gfCNCPoint6[12068] = {X 364.4434, Y 8.9212, Z -8.0000, A 0.000, B 0.000, C 0.000 }
gfCNCPoint6[12069] = {X 365.7826, Y 10.9065, Z -8.0000, A 0.000, B 0.000, C 0.000 }
gfCNCPoint6[12070] = {X 366.9214, Y 13.0132, Z -8.0000, A 0.000, B 0.000, C 0.000 }
gfCNCPoint6[12071] = {X 367.8488, Y 15.2212, Z -8.0000, A 0.000, B 0.000, C 0.000 }
gfCNCPoint6[12072] = {X 368.5559, Y 17.5092, Z -8.0000, A 0.000, B 0.000, C 0.000 }
gfCNCPoint6[12073] = {X 369.0331, Y 19.7784, Z -8.0000, A 0.000, B 0.000, C 0.000 }
gfCNCPoint6[12074] = {X 369.3408, Y 22.0767, Z -8.0000, A 0.000, B 0.000, C 0.000 }
gfCNCPoint6[12075] = {X 369.4773, Y 24.3915, Z -8.0000, A 0.000, B 0.000, C 0.000 }
gfCNCPoint6[12076] = {X 369.4418, Y 26.7100, Z -8.0000, A 0.000, B 0.000, C 0.000 }
gfCNCPoint6[12077] = {X 369.2346, Y 29.0196, Z -8.0000, A 0.000, B 0.000, C 0.000 }
gfCNCPoint6[12078] = {X 368.8568, Y 31.3074, Z -8.0000, A 0.000, B 0.000, C 0.000 }
gfCNCPoint6[12079] = {X 368.3394, Y 33.3846, Z -8.0000, A 0.000, B 0.000, C 0.000 }
gfCNCPoint6[12080] = {X 367.6406, Y 35.4079, Z -8.0000, A 0.000, B 0.000, C 0.000 }
gfCNCPoint6[12081] = {X 366.7658, Y 37.3616, Z -8.0000, A 0.000, B 0.000, C 0.000 }
gfCNCPoint6[12082] = {X 365.7220, Y 39.2305, Z -8.0000, A 0.000, B 0.000, C 0.000 }
gfCNCPoint6[12083] = {X 364.5172, Y 40.9999, Z -8.0000, A 0.000, B 0.000, C 0.000 }
gfCNCPoint6[12084] = {X 364.4579, Y 41.0809, Z -8.0000, A 0.000, B 0.000, C 0.000 }
gfCNCPoint6[12085] = {X 367.7503, Y 43.4906, Z -8.0000, A 0.000, B 0.000, C 0.000 }
gfCNCPoint6[12086] = {X 367.7503, Y 43.4906, Z -5.0000, A 0.000, B 0.000, C 0.000 }
gfCNCPoint6[12087] = {X 367.7503, Y 43.4906, Z 11.0000, A 0.000, B 0.000, C 0.000 }
gfCNCPoint6[12088] = {X 606.0426, Y 42.9003, Z 11.0000, A 0.000, B 0.000, C 0.000 }
gfCNCPoint6[12089] = {X 606.0426, Y 42.9003, Z -5.0000, A 0.000, B 0.000, C 0.000 }
gfCNCPoint6[12090] = {X 606.0426, Y 42.9003, Z -8.0000, A 0.000, B 0.000, C 0.000 }
gfCNCPoint6[12091] = {X 603.6967, Y 47.0765, Z -8.0000, A 0.000, B 0.000, C 0.000 }
gfCNCPoint6[12092] = {X 603.6312, Y 47.1891, Z -8.0000, A 0.000, B 0.000, C 0.000 }
gfCNCPoint6[12093] = {X 603.5623, Y 47.2995, Z -8.0000, A 0.000, B 0.000, C 0.000 }
gfCNCPoint6[12094] = {X 603.0359, Y 47.9599, Z -8.0000, A 0.000, B 0.000, C 0.000 }
gfCNCPoint6[12095] = {X 602.3890, Y 48.5029, Z -8.0000, A 0.000, B 0.000, C 0.000 }
gfCNCPoint6[12096] = {X 601.6473, Y 48.9069, Z -8.0000, A 0.000, B 0.000, C 0.000 }
gfCNCPoint6[12097] = {X 600.8403, Y 49.1559, Z -8.0000, A 0.000, B 0.000, C 0.000 }
gfCNCPoint6[12098] = {X 600.0000, Y 49.2400, Z -8.0000, A 0.000, B 0.000, C 0.000 }
gfCNCPoint6[12099] = {X 593.5565, Y 49.2400, Z -8.0000, A 0.000, B 0.000, C 0.000 }
gfCNCPoint6[12100] = {X 592.6130, Y 49.1337, Z -8.0000, A 0.000, B 0.000, C 0.000 }
gfCNCPoint6[12101] = {X 591.7169, Y 48.8201, Z -8.0000, A 0.000, B 0.000, C 0.000 }
gfCNCPoint6[12102] = {X 590.9129, Y 48.3150, Z -8.0000, A 0.000, B 0.000, C 0.000 }
gfCNCPoint6[12103] = {X 590.2416, Y 47.6436, Z -8.0000, A 0.000, B 0.000, C 0.000 }
gfCNCPoint6[12104] = {X 589.7364, Y 46.8397, Z -8.0000, A 0.000, B 0.000, C 0.000 }
gfCNCPoint6[12105] = {X 589.4228, Y 45.9435, Z -8.0000, A 0.000, B 0.000, C 0.000 }
gfCNCPoint6[12106] = {X 589.3165, Y 45.0000, Z -8.0000, A 0.000, B 0.000, C 0.000 }
gfCNCPoint6[12107] = {X 589.3165, Y 44.0651, Z -8.0000, A 0.000, B 0.000, C 0.000 }
gfCNCPoint6[12108] = {X 589.4202, Y 43.1448, Z -8.0000, A 0.000, B 0.000, C 0.000 }
gfCNCPoint6[12109] = {X 589.7196, Y 42.2684, Z -8.0000, A 0.000, B 0.000, C 0.000 }
gfCNCPoint6[12110] = {X 590.2007, Y 41.4770, Z -8.0000, A 0.000, B 0.000, C 0.000 }
gfCNCPoint6[12111] = {X 590.8409, Y 40.8078, Z -8.0000, A 0.000, B 0.000, C 0.000 }
gfCNCPoint6[12112] = {X 590.8418, Y 33.1230, Z -8.0000, A 0.000, B 0.000, C 0.000 }
gfCNCPoint6[12113] = {X 585.3714, Y 46.6218, Z -8.0000, A 0.000, B 0.000, C 0.000 }
gfCNCPoint6[12114] = {X 585.0085, Y 47.3114, Z -8.0000, A 0.000, B 0.000, C 0.000 }
gfCNCPoint6[12115] = {X 584.5255, Y 47.9228, Z -8.0000, A 0.000, B 0.000, C 0.000 }
gfCNCPoint6[12116] = {X 583.9387, Y 48.4356, Z -8.0000, A 0.000, B 0.000, C 0.000 }
gfCNCPoint6[12117] = {X 583.2680, Y 48.8323, Z -8.0000, A 0.000, B 0.000, C 0.000 }
gfCNCPoint6[12118] = {X 582.3418, Y 49.1460, Z -8.0000, A 0.000, B 0.000, C 0.000 }
gfCNCPoint6[12119] = {X 581.3682, Y 49.2391, Z -8.0000, A 0.000, B 0.000, C 0.000 }
gfCNCPoint6[12120] = {X 580.3993, Y 49.1068, Z -8.0000, A 0.000, B 0.000, C 0.000 }
gfCNCPoint6[12121] = {X 579.4864, Y 48.7559, Z -8.0000, A 0.000, B 0.000, C 0.000 }
gfCNCPoint6[12122] = {X 578.6782, Y 48.2052, Z -8.0000, A 0.000, B 0.000, C 0.000 }
gfCNCPoint6[12123] = {X 578.0177, Y 47.4840, Z -8.0000, A 0.000, B 0.000, C 0.000 }
gfCNCPoint6[12124] = {X 577.5400, Y 46.6307, Z -8.0000, A 0.000, B 0.000, C 0.000 }
gfCNCPoint6[12125] = {X 571.9402, Y 32.9378, Z -8.0000, A 0.000, B 0.000, C 0.000 }
gfCNCPoint6[12126] = {X 571.9404, Y 40.8087, Z -8.0000, A 0.000, B 0.000, C 0.000 }
gfCNCPoint6[12127] = {X 571.9716, Y 40.8346, Z -8.0000, A 0.000, B 0.000, C 0.000 }
gfCNCPoint6[12128] = {X 572.5965, Y 41.4929, Z -8.0000, A 0.000, B 0.000, C 0.000 }
gfCNCPoint6[12129] = {X 573.0669, Y 42.2692, Z -8.0000, A 0.000, B 0.000, C 0.000 }
gfCNCPoint6[12130] = {X 573.3613, Y 43.1278, Z -8.0000, A 0.000, B 0.000, C 0.000 }
gfCNCPoint6[12131] = {X 573.4663, Y 44.0294, Z -8.0000, A 0.000, B 0.000, C 0.000 }
gfCNCPoint6[12132] = {X 573.4664, Y 45.0000, Z -8.0000, A 0.000, B 0.000, C 0.000 }
gfCNCPoint6[12133] = {X 573.3601, Y 45.9435, Z -8.0000, A 0.000, B 0.000, C 0.000 }
gfCNCPoint6[12134] = {X 573.0465, Y 46.8397, Z -8.0000, A 0.000, B 0.000, C 0.000 }
gfCNCPoint6[12135] = {X 572.5414, Y 47.6436, Z -8.0000, A 0.000, B 0.000, C 0.000 }
gfCNCPoint6[12136] = {X 571.8700, Y 48.3150, Z -8.0000, A 0.000, B 0.000, C 0.000 }
gfCNCPoint6[12137] = {X 571.0661, Y 48.8201, Z -8.0000, A 0.000, B 0.000, C 0.000 }
gfCNCPoint6[12138] = {X 570.1699, Y 49.1337, Z -8.0000, A 0.000, B 0.000, C 0.000 }
gfCNCPoint6[12139] = {X 569.2264, Y 49.2400, Z -8.0000, A 0.000, B 0.000, C 0.000 }
gfCNCPoint6[12140] = {X 562.4443, Y 49.2400, Z -8.0000, A 0.000, B 0.000, C 0.000 }
gfCNCPoint6[12141] = {X 561.5008, Y 49.1337, Z -8.0000, A 0.000, B 0.000, C 0.000 }
gfCNCPoint6[12142] = {X 560.6046, Y 48.8201, Z -8.0000, A 0.000, B 0.000, C 0.000 }
gfCNCPoint6[12143] = {X 559.8007, Y 48.3150, Z -8.0000, A 0.000, B 0.000, C 0.000 }
gfCNCPoint6[12144] = {X 559.1293, Y 47.6436, Z -8.0000, A 0.000, B 0.000, C 0.000 }
gfCNCPoint6[12145] = {X 558.6242, Y 46.8397, Z -8.0000, A 0.000, B 0.000, C 0.000 }
gfCNCPoint6[12146] = {X 558.3106, Y 45.9435, Z -8.0000, A 0.000, B 0.000, C 0.000 }
gfCNCPoint6[12147] = {X 558.2043, Y 45.0000, Z -8.0000, A 0.000, B 0.000, C 0.000 }
gfCNCPoint6[12148] = {X 558.2043, Y 44.0652, Z -8.0000, A 0.000, B 0.000, C 0.000 }
gfCNCPoint6[12149] = {X 558.3078, Y 43.1444, Z -8.0000, A 0.000, B 0.000, C 0.000 }
gfCNCPoint6[12150] = {X 558.6075, Y 42.2677, Z -8.0000, A 0.000, B 0.000, C 0.000 }
gfCNCPoint6[12151] = {X 559.0893, Y 41.4762, Z -8.0000, A 0.000, B 0.000, C 0.000 }
gfCNCPoint6[12152] = {X 559.7306, Y 40.8074, Z -8.0000, A 0.000, B 0.000, C 0.000 }
gfCNCPoint6[12153] = {X 559.7310, Y 9.1922, Z -8.0000, A 0.000, B 0.000, C 0.000 }
gfCNCPoint6[12154] = {X 559.0934, Y 8.5319, Z -8.0000, A 0.000, B 0.000, C 0.000 }
gfCNCPoint6[12155] = {X 558.6128, Y 7.7499, Z -8.0000, A 0.000, B 0.000, C 0.000 }
gfCNCPoint6[12156] = {X 558.3118, Y 6.8827, Z -8.0000, A 0.000, B 0.000, C 0.000 }
gfCNCPoint6[12157] = {X 558.2045, Y 5.9711, Z -8.0000, A 0.000, B 0.000, C 0.000 }
gfCNCPoint6[12158] = {X 558.2043, Y 5.0000, Z -8.0000, A 0.000, B 0.000, C 0.000 }
gfCNCPoint6[12159] = {X 558.3106, Y 4.0565, Z -8.0000, A 0.000, B 0.000, C 0.000 }
gfCNCPoint6[12160] = {X 558.6242, Y 3.1603, Z -8.0000, A 0.000, B 0.000, C 0.000 }
gfCNCPoint6[12161] = {X 559.1293, Y 2.3564, Z -8.0000, A 0.000, B 0.000, C 0.000 }
gfCNCPoint6[12162] = {X 559.8007, Y 1.6850, Z -8.0000, A 0.000, B 0.000, C 0.000 }
gfCNCPoint6[12163] = {X 560.6046, Y 1.1799, Z -8.0000, A 0.000, B 0.000, C 0.000 }
gfCNCPoint6[12164] = {X 561.5008, Y 0.8663, Z -8.0000, A 0.000, B 0.000, C 0.000 }
gfCNCPoint6[12165] = {X 562.4443, Y 0.7600, Z -8.0000, A 0.000, B 0.000, C 0.000 }
gfCNCPoint6[12166] = {X 570.9376, Y 0.7600, Z -8.0000, A 0.000, B 0.000, C 0.000 }
gfCNCPoint6[12167] = {X 571.8810, Y 0.8663, Z -8.0000, A 0.000, B 0.000, C 0.000 }
gfCNCPoint6[12168] = {X 572.7772, Y 1.1799, Z -8.0000, A 0.000, B 0.000, C 0.000 }
gfCNCPoint6[12169] = {X 573.5812, Y 1.6850, Z -8.0000, A 0.000, B 0.000, C 0.000 }
gfCNCPoint6[12170] = {X 574.2525, Y 2.3564, Z -8.0000, A 0.000, B 0.000, C 0.000 }
gfCNCPoint6[12171] = {X 574.7577, Y 3.1603, Z -8.0000, A 0.000, B 0.000, C 0.000 }
gfCNCPoint6[12172] = {X 575.0712, Y 4.0565, Z -8.0000, A 0.000, B 0.000, C 0.000 }
gfCNCPoint6[12173] = {X 575.1776, Y 5.0000, Z -8.0000, A 0.000, B 0.000, C 0.000 }
gfCNCPoint6[12174] = {X 575.1776, Y 5.9343, Z -8.0000, A 0.000, B 0.000, C 0.000 }
gfCNCPoint6[12175] = {X 575.1024, Y 6.7286, Z -8.0000, A 0.000, B 0.000, C 0.000 }
gfCNCPoint6[12176] = {X 574.8798, Y 7.4948, Z -8.0000, A 0.000, B 0.000, C 0.000 }
gfCNCPoint6[12177] = {X 574.5176, Y 8.2058, Z -8.0000, A 0.000, B 0.000, C 0.000 }
gfCNCPoint6[12178] = {X 581.1908, Y 24.5801, Z -8.0000, A 0.000, B 0.000, C 0.000 }
gfCNCPoint6[12179] = {X 587.9344, Y 8.0873, Z -8.0000, A 0.000, B 0.000, C 0.000 }
gfCNCPoint6[12180] = {X 587.6157, Y 7.4195, Z -8.0000, A 0.000, B 0.000, C 0.000 }
gfCNCPoint6[12181] = {X 587.4179, Y 6.7064, Z -8.0000, A 0.000, B 0.000, C 0.000 }
gfCNCPoint6[12182] = {X 587.3471, Y 5.9698, Z -8.0000, A 0.000, B 0.000, C 0.000 }
gfCNCPoint6[12183] = {X 587.3470, Y 5.0000, Z -8.0000, A 0.000, B 0.000, C 0.000 }
gfCNCPoint6[12184] = {X 587.4533, Y 4.0565, Z -8.0000, A 0.000, B 0.000, C 0.000 }
gfCNCPoint6[12185] = {X 587.7668, Y 3.1603, Z -8.0000, A 0.000, B 0.000, C 0.000 }
gfCNCPoint6[12186] = {X 588.2720, Y 2.3564, Z -8.0000, A 0.000, B 0.000, C 0.000 }
gfCNCPoint6[12187] = {X 588.9434, Y 1.6850, Z -8.0000, A 0.000, B 0.000, C 0.000 }
gfCNCPoint6[12188] = {X 589.7473, Y 1.1799, Z -8.0000, A 0.000, B 0.000, C 0.000 }
gfCNCPoint6[12189] = {X 590.6435, Y 0.8663, Z -8.0000, A 0.000, B 0.000, C 0.000 }
gfCNCPoint6[12190] = {X 591.5870, Y 0.7600, Z -8.0000, A 0.000, B 0.000, C 0.000 }
gfCNCPoint6[12191] = {X 600.0000, Y 0.7600, Z -8.0000, A 0.000, B 0.000, C 0.000 }
gfCNCPoint6[12192] = {X 600.8403, Y 0.8441, Z -8.0000, A 0.000, B 0.000, C 0.000 }
gfCNCPoint6[12193] = {X 601.6473, Y 1.0931, Z -8.0000, A 0.000, B 0.000, C 0.000 }
gfCNCPoint6[12194] = {X 602.3890, Y 1.4971, Z -8.0000, A 0.000, B 0.000, C 0.000 }
gfCNCPoint6[12195] = {X 603.0359, Y 2.0401, Z -8.0000, A 0.000, B 0.000, C 0.000 }
gfCNCPoint6[12196] = {X 603.5623, Y 2.7005, Z -8.0000, A 0.000, B 0.000, C 0.000 }
gfCNCPoint6[12197] = {X 603.6312, Y 2.8109, Z -8.0000, A 0.000, B 0.000, C 0.000 }
gfCNCPoint6[12198] = {X 603.6967, Y 2.9235, Z -8.0000, A 0.000, B 0.000, C 0.000 }
gfCNCPoint6[12199] = {X 607.8224, Y 10.2681, Z -8.0000, A 0.000, B 0.000, C 0.000 }
gfCNCPoint6[12200] = {X 607.8224, Y 10.2681, Z -5.0000, A 0.000, B 0.000, C 0.000 }
gfCNCPoint6[12201] = {X 607.8224, Y 10.2681, Z 11.0000, A 0.000, B 0.000, C 0.000 }
gfCNCPoint6[12202] = {X 607.6967, Y 39.1575, Z 11.0000, A 0.000, B 0.000, C 0.000 }
gfCNCPoint6[12203] = {X 607.6967, Y 39.1575, Z -5.0000, A 0.000, B 0.000, C 0.000 }
gfCNCPoint6[12204] = {X 607.6967, Y 39.1575, Z -8.0000, A 0.000, B 0.000, C 0.000 }
gfCNCPoint6[12205] = {X 603.6967, Y 46.9079, Z -8.0000, A 0.000, B 0.000, C 0.000 }
gfCNCPoint6[12206] = {X 603.6001, Y 47.0845, Z -8.0000, A 0.000, B 0.000, C 0.000 }
gfCNCPoint6[12207] = {X 603.4951, Y 47.2561, Z -8.0000, A 0.000, B 0.000, C 0.000 }
gfCNCPoint6[12208] = {X 602.9786, Y 47.9041, Z -8.0000, A 0.000, B 0.000, C 0.000 }
gfCNCPoint6[12209] = {X 602.3439, Y 48.4368, Z -8.0000, A 0.000, B 0.000, C 0.000 }
gfCNCPoint6[12210] = {X 601.6163, Y 48.8332, Z -8.0000, A 0.000, B 0.000, C 0.000 }
gfCNCPoint6[12211] = {X 600.8245, Y 49.0775, Z -8.0000, A 0.000, B 0.000, C 0.000 }
gfCNCPoint6[12212] = {X 600.0000, Y 49.1600, Z -8.0000, A 0.000, B 0.000, C 0.000 }
gfCNCPoint6[12213] = {X 593.5565, Y 49.1600, Z -8.0000, A 0.000, B 0.000, C 0.000 }
gfCNCPoint6[12214] = {X 592.6308, Y 49.0557, Z -8.0000, A 0.000, B 0.000, C 0.000 }
gfCNCPoint6[12215] = {X 591.7516, Y 48.7480, Z -8.0000, A 0.000, B 0.000, C 0.000 }
gfCNCPoint6[12216] = {X 590.9628, Y 48.2524, Z -8.0000, A 0.000, B 0.000, C 0.000 }
gfCNCPoint6[12217] = {X 590.3041, Y 47.5937, Z -8.0000, A 0.000, B 0.000, C 0.000 }
gfCNCPoint6[12218] = {X 589.8085, Y 46.8050, Z -8.0000, A 0.000, B 0.000, C 0.000 }
gfCNCPoint6[12219] = {X 589.5008, Y 45.9257, Z -8.0000, A 0.000, B 0.000, C 0.000 }
gfCNCPoint6[12220] = {X 589.3965, Y 45.0000, Z -8.0000, A 0.000, B 0.000, C 0.000 }
gfCNCPoint6[12221] = {X 589.3965, Y 44.0654, Z -8.0000, A 0.000, B 0.000, C 0.000 }
gfCNCPoint6[12222] = {X 589.5003, Y 43.1532, Z -8.0000, A 0.000, B 0.000, C 0.000 }
gfCNCPoint6[12223] = {X 589.8000, Y 42.2855, Z -8.0000, A 0.000, B 0.000, C 0.000 }
gfCNCPoint6[12224] = {X 590.2812, Y 41.5037, Z -8.0000, A 0.000, B 0.000, C 0.000 }
gfCNCPoint6[12225] = {X 590.9209, Y 40.8452, Z -8.0000, A 0.000, B 0.000, C 0.000 }
gfCNCPoint6[12226] = {X 590.9218, Y 32.7125, Z -8.0000, A 0.000, B 0.000, C 0.000 }
gfCNCPoint6[12227] = {X 585.2975, Y 46.5912, Z -8.0000, A 0.000, B 0.000, C 0.000 }
gfCNCPoint6[12228] = {X 584.9414, Y 47.2678, Z -8.0000, A 0.000, B 0.000, C 0.000 }
gfCNCPoint6[12229] = {X 584.4675, Y 47.8677, Z -8.0000, A 0.000, B 0.000, C 0.000 }
gfCNCPoint6[12230] = {X 583.8918, Y 48.3708, Z -8.0000, A 0.000, B 0.000, C 0.000 }
gfCNCPoint6[12231] = {X 583.2338, Y 48.7600, Z -8.0000, A 0.000, B 0.000, C 0.000 }
gfCNCPoint6[12232] = {X 582.3250, Y 49.0678, Z -8.0000, A 0.000, B 0.000, C 0.000 }
gfCNCPoint6[12233] = {X 581.3699, Y 49.1592, Z -8.0000, A 0.000, B 0.000, C 0.000 }
gfCNCPoint6[12234] = {X 580.4192, Y 49.0293, Z -8.0000, A 0.000, B 0.000, C 0.000 }
gfCNCPoint6[12235] = {X 579.5236, Y 48.6850, Z -8.0000, A 0.000, B 0.000, C 0.000 }
gfCNCPoint6[12236] = {X 578.7306, Y 48.1448, Z -8.0000, A 0.000, B 0.000, C 0.000 }
gfCNCPoint6[12237] = {X 578.0826, Y 47.4372, Z -8.0000, A 0.000, B 0.000, C 0.000 }
gfCNCPoint6[12238] = {X 577.6138, Y 46.5999, Z -8.0000, A 0.000, B 0.000, C 0.000 }
gfCNCPoint6[12239] = {X 571.8602, Y 32.5308, Z -8.0000, A 0.000, B 0.000, C 0.000 }
gfCNCPoint6[12240] = {X 571.8604, Y 40.8463, Z -8.0000, A 0.000, B 0.000, C 0.000 }
gfCNCPoint6[12241] = {X 571.9201, Y 40.8958, Z -8.0000, A 0.000, B 0.000, C 0.000 }
gfCNCPoint6[12242] = {X 572.5331, Y 41.5417, Z -8.0000, A 0.000, B 0.000, C 0.000 }
gfCNCPoint6[12243] = {X 572.9945, Y 42.3033, Z -8.0000, A 0.000, B 0.000, C 0.000 }
gfCNCPoint6[12244] = {X 573.2834, Y 43.1456, Z -8.0000, A 0.000, B 0.000, C 0.000 }
gfCNCPoint6[12245] = {X 573.3863, Y 44.0301, Z -8.0000, A 0.000, B 0.000, C 0.000 }
gfCNCPoint6[12246] = {X 573.3864, Y 45.0000, Z -8.0000, A 0.000, B 0.000, C 0.000 }
gfCNCPoint6[12247] = {X 573.2821, Y 45.9257, Z -8.0000, A 0.000, B 0.000, C 0.000 }
gfCNCPoint6[12248] = {X 572.9745, Y 46.8050, Z -8.0000, A 0.000, B 0.000, C 0.000 }
gfCNCPoint6[12249] = {X 572.4788, Y 47.5937, Z -8.0000, A 0.000, B 0.000, C 0.000 }
gfCNCPoint6[12250] = {X 571.8201, Y 48.2524, Z -8.0000, A 0.000, B 0.000, C 0.000 }
gfCNCPoint6[12251] = {X 571.0314, Y 48.7480, Z -8.0000, A 0.000, B 0.000, C 0.000 }
gfCNCPoint6[12252] = {X 570.1521, Y 49.0557, Z -8.0000, A 0.000, B 0.000, C 0.000 }
gfCNCPoint6[12253] = {X 569.2264, Y 49.1600, Z -8.0000, A 0.000, B 0.000, C 0.000 }
gfCNCPoint6[12254] = {X 562.4443, Y 49.1600, Z -8.0000, A 0.000, B 0.000, C 0.000 }
gfCNCPoint6[12255] = {X 561.5186, Y 49.0557, Z -8.0000, A 0.000, B 0.000, C 0.000 }
gfCNCPoint6[12256] = {X 560.6393, Y 48.7480, Z -8.0000, A 0.000, B 0.000, C 0.000 }
gfCNCPoint6[12257] = {X 559.8506, Y 48.2524, Z -8.0000, A 0.000, B 0.000, C 0.000 }
gfCNCPoint6[12258] = {X 559.1919, Y 47.5937, Z -8.0000, A 0.000, B 0.000, C 0.000 }
gfCNCPoint6[12259] = {X 558.6963, Y 46.8050, Z -8.0000, A 0.000, B 0.000, C 0.000 }
gfCNCPoint6[12260] = {X 558.3886, Y 45.9257, Z -8.0000, A 0.000, B 0.000, C 0.000 }
gfCNCPoint6[12261] = {X 558.2843, Y 45.0000, Z -8.0000, A 0.000, B 0.000, C 0.000 }
gfCNCPoint6[12262] = {X 558.2843, Y 44.0655, Z -8.0000, A 0.000, B 0.000, C 0.000 }
gfCNCPoint6[12263] = {X 558.3879, Y 43.1529, Z -8.0000, A 0.000, B 0.000, C 0.000 }
gfCNCPoint6[12264] = {X 558.6878, Y 42.2848, Z -8.0000, A 0.000, B 0.000, C 0.000 }
gfCNCPoint6[12265] = {X 559.1698, Y 41.5029, Z -8.0000, A 0.000, B 0.000, C 0.000 }
gfCNCPoint6[12266] = {X 559.8106, Y 40.8449, Z -8.0000, A 0.000, B 0.000, C 0.000 }
gfCNCPoint6[12267] = {X 559.8110, Y 9.1545, Z -8.0000, A 0.000, B 0.000, C 0.000 }
gfCNCPoint6[12268] = {X 559.1738, Y 8.5050, Z -8.0000, A 0.000, B 0.000, C 0.000 }
gfCNCPoint6[12269] = {X 558.6931, Y 7.7325, Z -8.0000, A 0.000, B 0.000, C 0.000 }
gfCNCPoint6[12270] = {X 558.3919, Y 6.8739, Z -8.0000, A 0.000, B 0.000, C 0.000 }
gfCNCPoint6[12271] = {X 558.2845, Y 5.9704, Z -8.0000, A 0.000, B 0.000, C 0.000 }
gfCNCPoint6[12272] = {X 558.2843, Y 5.0000, Z -8.0000, A 0.000, B 0.000, C 0.000 }
gfCNCPoint6[12273] = {X 558.3886, Y 4.0743, Z -8.0000, A 0.000, B 0.000, C 0.000 }
gfCNCPoint6[12274] = {X 558.6963, Y 3.1950, Z -8.0000, A 0.000, B 0.000, C 0.000 }
gfCNCPoint6[12275] = {X 559.1919, Y 2.4063, Z -8.0000, A 0.000, B 0.000, C 0.000 }
gfCNCPoint6[12276] = {X 559.8506, Y 1.7476, Z -8.0000, A 0.000, B 0.000, C 0.000 }
gfCNCPoint6[12277] = {X 560.6393, Y 1.2520, Z -8.0000, A 0.000, B 0.000, C 0.000 }
gfCNCPoint6[12278] = {X 561.5186, Y 0.9443, Z -8.0000, A 0.000, B 0.000, C 0.000 }
gfCNCPoint6[12279] = {X 562.4443, Y 0.8400, Z -8.0000, A 0.000, B 0.000, C 0.000 }
gfCNCPoint6[12280] = {X 570.9376, Y 0.8400, Z -8.0000, A 0.000, B 0.000, C 0.000 }
gfCNCPoint6[12281] = {X 571.8632, Y 0.9443, Z -8.0000, A 0.000, B 0.000, C 0.000 }
gfCNCPoint6[12282] = {X 572.7425, Y 1.2520, Z -8.0000, A 0.000, B 0.000, C 0.000 }
gfCNCPoint6[12283] = {X 573.5313, Y 1.7476, Z -8.0000, A 0.000, B 0.000, C 0.000 }
gfCNCPoint6[12284] = {X 574.1900, Y 2.4063, Z -8.0000, A 0.000, B 0.000, C 0.000 }
gfCNCPoint6[12285] = {X 574.6856, Y 3.1950, Z -8.0000, A 0.000, B 0.000, C 0.000 }
gfCNCPoint6[12286] = {X 574.9933, Y 4.0743, Z -8.0000, A 0.000, B 0.000, C 0.000 }
gfCNCPoint6[12287] = {X 575.0976, Y 5.0000, Z -8.0000, A 0.000, B 0.000, C 0.000 }
gfCNCPoint6[12288] = {X 575.0976, Y 5.9343, Z -8.0000, A 0.000, B 0.000, C 0.000 }
gfCNCPoint6[12289] = {X 575.0213, Y 6.7271, Z -8.0000, A 0.000, B 0.000, C 0.000 }
gfCNCPoint6[12290] = {X 574.7953, Y 7.4908, Z -8.0000, A 0.000, B 0.000, C 0.000 }
gfCNCPoint6[12291] = {X 574.4279, Y 8.1975, Z -8.0000, A 0.000, B 0.000, C 0.000 }
gfCNCPoint6[12292] = {X 581.1907, Y 24.7918, Z -8.0000, A 0.000, B 0.000, C 0.000 }
gfCNCPoint6[12293] = {X 588.0236, Y 8.0807, Z -8.0000, A 0.000, B 0.000, C 0.000 }
gfCNCPoint6[12294] = {X 587.6999, Y 7.4161, Z -8.0000, A 0.000, B 0.000, C 0.000 }
gfCNCPoint6[12295] = {X 587.4990, Y 6.7048, Z -8.0000, A 0.000, B 0.000, C 0.000 }
gfCNCPoint6[12296] = {X 587.4271, Y 5.9692, Z -8.0000, A 0.000, B 0.000, C 0.000 }
gfCNCPoint6[12297] = {X 587.4270, Y 5.0000, Z -8.0000, A 0.000, B 0.000, C 0.000 }
gfCNCPoint6[12298] = {X 587.5313, Y 4.0743, Z -8.0000, A 0.000, B 0.000, C 0.000 }
gfCNCPoint6[12299] = {X 587.8389, Y 3.1950, Z -8.0000, A 0.000, B 0.000, C 0.000 }
gfCNCPoint6[12300] = {X 588.3345, Y 2.4063, Z -8.0000, A 0.000, B 0.000, C 0.000 }
gfCNCPoint6[12301] = {X 588.9932, Y 1.7476, Z -8.0000, A 0.000, B 0.000, C 0.000 }
gfCNCPoint6[12302] = {X 589.7820, Y 1.2520, Z -8.0000, A 0.000, B 0.000, C 0.000 }
gfCNCPoint6[12303] = {X 590.6613, Y 0.9443, Z -8.0000, A 0.000, B 0.000, C 0.000 }
gfCNCPoint6[12304] = {X 591.5870, Y 0.8400, Z -8.0000, A 0.000, B 0.000, C 0.000 }
gfCNCPoint6[12305] = {X 600.0000, Y 0.8400, Z -8.0000, A 0.000, B 0.000, C 0.000 }
gfCNCPoint6[12306] = {X 600.8245, Y 0.9225, Z -8.0000, A 0.000, B 0.000, C 0.000 }
gfCNCPoint6[12307] = {X 601.6163, Y 1.1668, Z -8.0000, A 0.000, B 0.000, C 0.000 }
gfCNCPoint6[12308] = {X 602.3439, Y 1.5632, Z -8.0000, A 0.000, B 0.000, C 0.000 }
gfCNCPoint6[12309] = {X 602.9786, Y 2.0959, Z -8.0000, A 0.000, B 0.000, C 0.000 }
gfCNCPoint6[12310] = {X 603.4951, Y 2.7439, Z -8.0000, A 0.000, B 0.000, C 0.000 }
gfCNCPoint6[12311] = {X 603.6001, Y 2.9155, Z -8.0000, A 0.000, B 0.000, C 0.000 }
gfCNCPoint6[12312] = {X 603.6967, Y 3.0921, Z -8.0000, A 0.000, B 0.000, C 0.000 }
gfCNCPoint6[12313] = {X 607.6967, Y 10.8425, Z -8.0000, A 0.000, B 0.000, C 0.000 }
gfCNCPoint6[12314] = {X 607.6967, Y 10.8425, Z -5.0000, A 0.000, B 0.000, C 0.000 }
gfCNCPoint6[12315] = {X 607.6967, Y 10.8425, Z 11.0000, A 0.000, B 0.000, C 0.000 }
gfCNCPoint6[12316] = {X 607.6967, Y 38.1620, Z 11.0000, A 0.000, B 0.000, C 0.000 }
gfCNCPoint6[12317] = {X 607.6967, Y 38.1620, Z -5.0000, A 0.000, B 0.000, C 0.000 }
gfCNCPoint6[12318] = {X 607.6967, Y 38.1620, Z -8.0000, A 0.000, B 0.000, C 0.000 }
gfCNCPoint6[12319] = {X 603.6967, Y 46.7265, Z -8.0000, A 0.000, B 0.000, C 0.000 }
gfCNCPoint6[12320] = {X 603.5706, Y 46.9742, Z -8.0000, A 0.000, B 0.000, C 0.000 }
gfCNCPoint6[12321] = {X 603.4278, Y 47.2128, Z -8.0000, A 0.000, B 0.000, C 0.000 }
gfCNCPoint6[12322] = {X 602.9213, Y 47.8482, Z -8.0000, A 0.000, B 0.000, C 0.000 }
gfCNCPoint6[12323] = {X 602.2988, Y 48.3707, Z -8.0000, A 0.000, B 0.000, C 0.000 }
gfCNCPoint6[12324] = {X 601.5852, Y 48.7595, Z -8.0000, A 0.000, B 0.000, C 0.000 }
gfCNCPoint6[12325] = {X 600.8086, Y 48.9991, Z -8.0000, A 0.000, B 0.000, C 0.000 }
gfCNCPoint6[12326] = {X 600.0000, Y 49.0800, Z -8.0000, A 0.000, B 0.000, C 0.000 }
gfCNCPoint6[12327] = {X 593.5565, Y 49.0800, Z -8.0000, A 0.000, B 0.000, C 0.000 }
gfCNCPoint6[12328] = {X 592.6486, Y 48.9777, Z -8.0000, A 0.000, B 0.000, C 0.000 }
gfCNCPoint6[12329] = {X 591.7863, Y 48.6760, Z -8.0000, A 0.000, B 0.000, C 0.000 }
gfCNCPoint6[12330] = {X 591.0127, Y 48.1899, Z -8.0000, A 0.000, B 0.000, C 0.000 }
gfCNCPoint6[12331] = {X 590.3667, Y 47.5438, Z -8.0000, A 0.000, B 0.000, C 0.000 }
gfCNCPoint6[12332] = {X 589.8806, Y 46.7702, Z -8.0000, A 0.000, B 0.000, C 0.000 }
gfCNCPoint6[12333] = {X 589.5788, Y 45.9079, Z -8.0000, A 0.000, B 0.000, C 0.000 }
gfCNCPoint6[12334] = {X 589.4765, Y 45.0000, Z -8.0000, A 0.000, B 0.000, C 0.000 }
gfCNCPoint6[12335] = {X 589.4765, Y 44.0657, Z -8.0000, A 0.000, B 0.000, C 0.000 }
gfCNCPoint6[12336] = {X 589.5726, Y 43.1968, Z -8.0000, A 0.000, B 0.000, C 0.000 }
gfCNCPoint6[12337] = {X 589.8499, Y 42.3678, Z -8.0000, A 0.000, B 0.000, C 0.000 }
gfCNCPoint6[12338] = {X 590.2961, Y 41.6161, Z -8.0000, A 0.000, B 0.000, C 0.000 }
gfCNCPoint6[12339] = {X 590.8909, Y 40.9755, Z -8.0000, A 0.000, B 0.000, C 0.000 }
gfCNCPoint6[12340] = {X 590.9455, Y 40.9288, Z -8.0000, A 0.000, B 0.000, C 0.000 }
gfCNCPoint6[12341] = {X 591.0009, Y 40.8832, Z -8.0000, A 0.000, B 0.000, C 0.000 }
gfCNCPoint6[12342] = {X 591.0019, Y 32.3019, Z -8.0000, A 0.000, B 0.000, C 0.000 }
gfCNCPoint6[12343] = {X 585.2236, Y 46.5606, Z -8.0000, A 0.000, B 0.000, C 0.000 }
gfCNCPoint6[12344] = {X 584.8743, Y 47.2242, Z -8.0000, A 0.000, B 0.000, C 0.000 }
gfCNCPoint6[12345] = {X 584.4095, Y 47.8125, Z -8.0000, A 0.000, B 0.000, C 0.000 }
gfCNCPoint6[12346] = {X 583.8449, Y 48.3059, Z -8.0000, A 0.000, B 0.000, C 0.000 }
gfCNCPoint6[12347] = {X 583.1996, Y 48.6877, Z -8.0000, A 0.000, B 0.000, C 0.000 }
gfCNCPoint6[12348] = {X 582.3082, Y 48.9895, Z -8.0000, A 0.000, B 0.000, C 0.000 }
gfCNCPoint6[12349] = {X 581.3715, Y 49.0792, Z -8.0000, A 0.000, B 0.000, C 0.000 }
gfCNCPoint6[12350] = {X 580.4391, Y 48.9518, Z -8.0000, A 0.000, B 0.000, C 0.000 }
gfCNCPoint6[12351] = {X 579.5607, Y 48.6142, Z -8.0000, A 0.000, B 0.000, C 0.000 }
gfCNCPoint6[12352] = {X 578.7830, Y 48.0843, Z -8.0000, A 0.000, B 0.000, C 0.000 }
gfCNCPoint6[12353] = {X 578.1474, Y 47.3903, Z -8.0000, A 0.000, B 0.000, C 0.000 }
gfCNCPoint6[12354] = {X 577.6877, Y 46.5692, Z -8.0000, A 0.000, B 0.000, C 0.000 }
gfCNCPoint6[12355] = {X 571.7802, Y 32.1238, Z -8.0000, A 0.000, B 0.000, C 0.000 }
gfCNCPoint6[12356] = {X 571.7804, Y 40.8839, Z -8.0000, A 0.000, B 0.000, C 0.000 }
gfCNCPoint6[12357] = {X 571.8687, Y 40.9571, Z -8.0000, A 0.000, B 0.000, C 0.000 }
gfCNCPoint6[12358] = {X 572.4697, Y 41.5906, Z -8.0000, A 0.000, B 0.000, C 0.000 }
gfCNCPoint6[12359] = {X 572.9222, Y 42.3374, Z -8.0000, A 0.000, B 0.000, C 0.000 }
gfCNCPoint6[12360] = {X 573.2054, Y 43.1634, Z -8.0000, A 0.000, B 0.000, C 0.000 }
gfCNCPoint6[12361] = {X 573.3063, Y 44.0308, Z -8.0000, A 0.000, B 0.000, C 0.000 }
gfCNCPoint6[12362] = {X 573.3064, Y 45.0000, Z -8.0000, A 0.000, B 0.000, C 0.000 }
gfCNCPoint6[12363] = {X 573.2041, Y 45.9079, Z -8.0000, A 0.000, B 0.000, C 0.000 }
gfCNCPoint6[12364] = {X 572.9024, Y 46.7702, Z -8.0000, A 0.000, B 0.000, C 0.000 }
gfCNCPoint6[12365] = {X 572.4163, Y 47.5438, Z -8.0000, A 0.000, B 0.000, C 0.000 }
gfCNCPoint6[12366] = {X 571.7703, Y 48.1899, Z -8.0000, A 0.000, B 0.000, C 0.000 }
gfCNCPoint6[12367] = {X 570.9967, Y 48.6760, Z -8.0000, A 0.000, B 0.000, C 0.000 }
gfCNCPoint6[12368] = {X 570.1343, Y 48.9777, Z -8.0000, A 0.000, B 0.000, C 0.000 }
gfCNCPoint6[12369] = {X 569.2264, Y 49.0800, Z -8.0000, A 0.000, B 0.000, C 0.000 }
gfCNCPoint6[12370] = {X 562.4443, Y 49.0800, Z -8.0000, A 0.000, B 0.000, C 0.000 }
gfCNCPoint6[12371] = {X 561.5364, Y 48.9777, Z -8.0000, A 0.000, B 0.000, C 0.000 }
gfCNCPoint6[12372] = {X 560.6741, Y 48.6760, Z -8.0000, A 0.000, B 0.000, C 0.000 }
gfCNCPoint6[12373] = {X 559.9005, Y 48.1899, Z -8.0000, A 0.000, B 0.000, C 0.000 }
gfCNCPoint6[12374] = {X 559.2544, Y 47.5438, Z -8.0000, A 0.000, B 0.000, C 0.000 }
gfCNCPoint6[12375] = {X 558.7683, Y 46.7702, Z -8.0000, A 0.000, B 0.000, C 0.000 }
gfCNCPoint6[12376] = {X 558.4666, Y 45.9079, Z -8.0000, A 0.000, B 0.000, C 0.000 }
gfCNCPoint6[12377] = {X 558.3643, Y 45.0000, Z -8.0000, A 0.000, B 0.000, C 0.000 }
gfCNCPoint6[12378] = {X 558.3643, Y 44.0657, Z -8.0000, A 0.000, B 0.000, C 0.000 }
gfCNCPoint6[12379] = {X 558.4601, Y 43.1965, Z -8.0000, A 0.000, B 0.000, C 0.000 }
gfCNCPoint6[12380] = {X 558.7377, Y 42.3672, Z -8.0000, A 0.000, B 0.000, C 0.000 }
gfCNCPoint6[12381] = {X 559.1845, Y 41.6154, Z -8.0000, A 0.000, B 0.000, C 0.000 }
gfCNCPoint6[12382] = {X 559.7803, Y 40.9753, Z -8.0000, A 0.000, B 0.000, C 0.000 }
gfCNCPoint6[12383] = {X 559.8350, Y 40.9286, Z -8.0000, A 0.000, B 0.000, C 0.000 }
gfCNCPoint6[12384] = {X 559.8906, Y 40.8829, Z -8.0000, A 0.000, B 0.000, C 0.000 }
gfCNCPoint6[12385] = {X 559.8910, Y 9.1164, Z -8.0000, A 0.000, B 0.000, C 0.000 }
gfCNCPoint6[12386] = {X 559.2543, Y 8.4778, Z -8.0000, A 0.000, B 0.000, C 0.000 }
gfCNCPoint6[12387] = {X 558.7735, Y 7.7149, Z -8.0000, A 0.000, B 0.000, C 0.000 }
gfCNCPoint6[12388] = {X 558.4719, Y 6.8651, Z -8.0000, A 0.000, B 0.000, C 0.000 }
gfCNCPoint6[12389] = {X 558.3645, Y 5.9697, Z -8.0000, A 0.000, B 0.000, C 0.000 }
gfCNCPoint6[12390] = {X 558.3643, Y 5.0000, Z -8.0000, A 0.000, B 0.000, C 0.000 }
gfCNCPoint6[12391] = {X 558.4666, Y 4.0921, Z -8.0000, A 0.000, B 0.000, C 0.000 }
gfCNCPoint6[12392] = {X 558.7683, Y 3.2298, Z -8.0000, A 0.000, B 0.000, C 0.000 }
gfCNCPoint6[12393] = {X 559.2544, Y 2.4562, Z -8.0000, A 0.000, B 0.000, C 0.000 }
gfCNCPoint6[12394] = {X 559.9005, Y 1.8101, Z -8.0000, A 0.000, B 0.000, C 0.000 }
gfCNCPoint6[12395] = {X 560.6741, Y 1.3240, Z -8.0000, A 0.000, B 0.000, C 0.000 }
gfCNCPoint6[12396] = {X 561.5364, Y 1.0223, Z -8.0000, A 0.000, B 0.000, C 0.000 }
gfCNCPoint6[12397] = {X 562.4443, Y 0.9200, Z -8.0000, A 0.000, B 0.000, C 0.000 }
gfCNCPoint6[12398] = {X 570.9376, Y 0.9200, Z -8.0000, A 0.000, B 0.000, C 0.000 }
gfCNCPoint6[12399] = {X 571.8454, Y 1.0223, Z -8.0000, A 0.000, B 0.000, C 0.000 }
gfCNCPoint6[12400] = {X 572.7078, Y 1.3240, Z -8.0000, A 0.000, B 0.000, C 0.000 }
gfCNCPoint6[12401] = {X 573.4814, Y 1.8101, Z -8.0000, A 0.000, B 0.000, C 0.000 }
gfCNCPoint6[12402] = {X 574.1274, Y 2.4562, Z -8.0000, A 0.000, B 0.000, C 0.000 }
gfCNCPoint6[12403] = {X 574.6135, Y 3.2298, Z -8.0000, A 0.000, B 0.000, C 0.000 }
gfCNCPoint6[12404] = {X 574.9153, Y 4.0921, Z -8.0000, A 0.000, B 0.000, C 0.000 }
gfCNCPoint6[12405] = {X 575.0176, Y 5.0000, Z -8.0000, A 0.000, B 0.000, C 0.000 }
gfCNCPoint6[12406] = {X 575.0176, Y 5.9343, Z -8.0000, A 0.000, B 0.000, C 0.000 }
gfCNCPoint6[12407] = {X 574.9501, Y 6.6731, Z -8.0000, A 0.000, B 0.000, C 0.000 }
gfCNCPoint6[12408] = {X 574.7499, Y 7.3875, Z -8.0000, A 0.000, B 0.000, C 0.000 }
gfCNCPoint6[12409] = {X 574.4236, Y 8.0539, Z -8.0000, A 0.000, B 0.000, C 0.000 }
gfCNCPoint6[12410] = {X 574.3792, Y 8.1253, Z -8.0000, A 0.000, B 0.000, C 0.000 }
gfCNCPoint6[12411] = {X 574.3333, Y 8.1958, Z -8.0000, A 0.000, B 0.000, C 0.000 }
gfCNCPoint6[12412] = {X 574.3601, Y 8.2421, Z -8.0000, A 0.000, B 0.000, C 0.000 }
gfCNCPoint6[12413] = {X 581.1906, Y 25.0035, Z -8.0000, A 0.000, B 0.000, C 0.000 }
gfCNCPoint6[12414] = {X 588.1129, Y 8.0736, Z -8.0000, A 0.000, B 0.000, C 0.000 }
gfCNCPoint6[12415] = {X 588.0734, Y 8.0081, Z -8.0000, A 0.000, B 0.000, C 0.000 }
gfCNCPoint6[12416] = {X 588.0352, Y 7.9419, Z -8.0000, A 0.000, B 0.000, C 0.000 }
gfCNCPoint6[12417] = {X 587.7485, Y 7.3171, Z -8.0000, A 0.000, B 0.000, C 0.000 }
gfCNCPoint6[12418] = {X 587.5708, Y 6.6530, Z -8.0000, A 0.000, B 0.000, C 0.000 }
gfCNCPoint6[12419] = {X 587.5071, Y 5.9685, Z -8.0000, A 0.000, B 0.000, C 0.000 }
gfCNCPoint6[12420] = {X 587.5070, Y 5.0000, Z -8.0000, A 0.000, B 0.000, C 0.000 }
gfCNCPoint6[12421] = {X 587.6092, Y 4.0921, Z -8.0000, A 0.000, B 0.000, C 0.000 }
gfCNCPoint6[12422] = {X 587.9110, Y 3.2298, Z -8.0000, A 0.000, B 0.000, C 0.000 }
gfCNCPoint6[12423] = {X 588.3971, Y 2.4562, Z -8.0000, A 0.000, B 0.000, C 0.000 }
gfCNCPoint6[12424] = {X 589.0431, Y 1.8101, Z -8.0000, A 0.000, B 0.000, C 0.000 }
gfCNCPoint6[12425] = {X 589.8167, Y 1.3240, Z -8.0000, A 0.000, B 0.000, C 0.000 }
gfCNCPoint6[12426] = {X 590.6791, Y 1.0223, Z -8.0000, A 0.000, B 0.000, C 0.000 }
gfCNCPoint6[12427] = {X 591.5870, Y 0.9200, Z -8.0000, A 0.000, B 0.000, C 0.000 }
gfCNCPoint6[12428] = {X 600.0000, Y 0.9200, Z -8.0000, A 0.000, B 0.000, C 0.000 }
gfCNCPoint6[12429] = {X 600.8086, Y 1.0009, Z -8.0000, A 0.000, B 0.000, C 0.000 }
gfCNCPoint6[12430] = {X 601.5852, Y 1.2405, Z -8.0000, A 0.000, B 0.000, C 0.000 }
gfCNCPoint6[12431] = {X 602.2988, Y 1.6293, Z -8.0000, A 0.000, B 0.000, C 0.000 }
gfCNCPoint6[12432] = {X 602.9213, Y 2.1518, Z -8.0000, A 0.000, B 0.000, C 0.000 }
gfCNCPoint6[12433] = {X 603.4278, Y 2.7872, Z -8.0000, A 0.000, B 0.000, C 0.000 }
gfCNCPoint6[12434] = {X 603.5706, Y 3.0258, Z -8.0000, A 0.000, B 0.000, C 0.000 }
gfCNCPoint6[12435] = {X 603.6967, Y 3.2735, Z -8.0000, A 0.000, B 0.000, C 0.000 }
gfCNCPoint6[12436] = {X 607.6967, Y 11.8380, Z -8.0000, A 0.000, B 0.000, C 0.000 }
gfCNCPoint6[12437] = {X 607.6967, Y 11.8380, Z -5.0000, A 0.000, B 0.000, C 0.000 }
gfCNCPoint6[12438] = {X 607.6967, Y 11.8380, Z 11.0000, A 0.000, B 0.000, C 0.000 }
gfCNCPoint6[12439] = {X 607.6967, Y 36.8500, Z 11.0000, A 0.000, B 0.000, C 0.000 }
gfCNCPoint6[12440] = {X 607.6967, Y 36.8500, Z -5.0000, A 0.000, B 0.000, C 0.000 }
gfCNCPoint6[12441] = {X 607.6967, Y 36.8500, Z -8.0000, A 0.000, B 0.000, C 0.000 }
gfCNCPoint6[12442] = {X 603.6967, Y 46.5279, Z -8.0000, A 0.000, B 0.000, C 0.000 }
gfCNCPoint6[12443] = {X 603.5432, Y 46.8562, Z -8.0000, A 0.000, B 0.000, C 0.000 }
gfCNCPoint6[12444] = {X 603.3606, Y 47.1694, Z -8.0000, A 0.000, B 0.000, C 0.000 }
gfCNCPoint6[12445] = {X 602.8640, Y 47.7924, Z -8.0000, A 0.000, B 0.000, C 0.000 }
gfCNCPoint6[12446] = {X 602.2538, Y 48.3046, Z -8.0000, A 0.000, B 0.000, C 0.000 }
gfCNCPoint6[12447] = {X 601.5541, Y 48.6858, Z -8.0000, A 0.000, B 0.000, C 0.000 }
gfCNCPoint6[12448] = {X 600.7928, Y 48.9207, Z -8.0000, A 0.000, B 0.000, C 0.000 }
gfCNCPoint6[12449] = {X 600.0000, Y 49.0000, Z -8.0000, A 0.000, B 0.000, C 0.000 }
gfCNCPoint6[12450] = {X 593.5565, Y 49.0000, Z -8.0000, A 0.000, B 0.000, C 0.000 }
gfCNCPoint6[12451] = {X 592.6664, Y 48.8997, Z -8.0000, A 0.000, B 0.000, C 0.000 }
gfCNCPoint6[12452] = {X 591.8210, Y 48.6039, Z -8.0000, A 0.000, B 0.000, C 0.000 }
gfCNCPoint6[12453] = {X 591.0626, Y 48.1273, Z -8.0000, A 0.000, B 0.000, C 0.000 }
gfCNCPoint6[12454] = {X 590.4292, Y 47.4940, Z -8.0000, A 0.000, B 0.000, C 0.000 }
gfCNCPoint6[12455] = {X 589.9527, Y 46.7355, Z -8.0000, A 0.000, B 0.000, C 0.000 }
gfCNCPoint6[12456] = {X 589.6568, Y 45.8901, Z -8.0000, A 0.000, B 0.000, C 0.000 }
gfCNCPoint6[12457] = {X 589.5565, Y 45.0000, Z -8.0000, A 0.000, B 0.000, C 0.000 }
gfCNCPoint6[12458] = {X 589.5565, Y 44.0660, Z -8.0000, A 0.000, B 0.000, C 0.000 }
gfCNCPoint6[12459] = {X 589.6507, Y 43.2140, Z -8.0000, A 0.000, B 0.000, C 0.000 }
gfCNCPoint6[12460] = {X 589.9227, Y 42.4011, Z -8.0000, A 0.000, B 0.000, C 0.000 }
gfCNCPoint6[12461] = {X 590.3602, Y 41.6640, Z -8.0000, A 0.000, B 0.000, C 0.000 }
gfCNCPoint6[12462] = {X 590.9434, Y 41.0358, Z -8.0000, A 0.000, B 0.000, C 0.000 }
gfCNCPoint6[12463] = {X 591.0115, Y 40.9779, Z -8.0000, A 0.000, B 0.000, C 0.000 }
gfCNCPoint6[12464] = {X 591.0808, Y 40.9215, Z -8.0000, A 0.000, B 0.000, C 0.000 }
gfCNCPoint6[12465] = {X 591.0819, Y 32.0443, Z -8.0000, A 0.000, B 0.000, C 0.000 }
gfCNCPoint6[12466] = {X 590.9675, Y 32.1736, Z -8.0000, A 0.000, B 0.000, C 0.000 }
gfCNCPoint6[12467] = {X 590.3109, Y 33.7939, Z -8.0000, A 0.000, B 0.000, C 0.000 }
gfCNCPoint6[12468] = {X 585.1497, Y 46.5300, Z -8.0000, A 0.000, B 0.000, C 0.000 }
gfCNCPoint6[12469] = {X 584.8073, Y 47.1805, Z -8.0000, A 0.000, B 0.000, C 0.000 }
gfCNCPoint6[12470] = {X 584.3516, Y 47.7574, Z -8.0000, A 0.000, B 0.000, C 0.000 }
gfCNCPoint6[12471] = {X 583.7980, Y 48.2411, Z -8.0000, A 0.000, B 0.000, C 0.000 }
gfCNCPoint6[12472] = {X 583.1653, Y 48.6154, Z -8.0000, A 0.000, B 0.000, C 0.000 }
gfCNCPoint6[12473] = {X 582.2878, Y 48.9121, Z -8.0000, A 0.000, B 0.000, C 0.000 }
gfCNCPoint6[12474] = {X 581.3656, Y 48.9990, Z -8.0000, A 0.000, B 0.000, C 0.000 }
gfCNCPoint6[12475] = {X 580.4481, Y 48.8715, Z -8.0000, A 0.000, B 0.000, C 0.000 }
gfCNCPoint6[12476] = {X 579.5845, Y 48.5363, Z -8.0000, A 0.000, B 0.000, C 0.000 }
gfCNCPoint6[12477] = {X 578.8212, Y 48.0115, Z -8.0000, A 0.000, B 0.000, C 0.000 }
gfCNCPoint6[12478] = {X 578.1990, Y 47.3251, Z -8.0000, A 0.000, B 0.000, C 0.000 }
gfCNCPoint6[12479] = {X 577.7515, Y 46.5141, Z -8.0000, A 0.000, B 0.000, C 0.000 }
gfCNCPoint6[12480] = {X 571.7002, Y 31.7168, Z -8.0000, A 0.000, B 0.000, C 0.000 }
gfCNCPoint6[12481] = {X 571.7004, Y 40.9215, Z -8.0000, A 0.000, B 0.000, C 0.000 }
gfCNCPoint6[12482] = {X 571.8391, Y 41.0371, Z -8.0000, A 0.000, B 0.000, C 0.000 }
gfCNCPoint6[12483] = {X 572.4246, Y 41.6635, Z -8.0000, A 0.000, B 0.000, C 0.000 }
gfCNCPoint6[12484] = {X 572.8631, Y 42.4002, Z -8.0000, A 0.000, B 0.000, C 0.000 }
gfCNCPoint6[12485] = {X 573.1345, Y 43.2135, Z -8.0000, A 0.000, B 0.000, C 0.000 }
gfCNCPoint6[12486] = {X 573.2264, Y 44.0660, Z -8.0000, A 0.000, B 0.000, C 0.000 }
gfCNCPoint6[12487] = {X 573.2264, Y 45.0000, Z -8.0000, A 0.000, B 0.000, C 0.000 }
gfCNCPoint6[12488] = {X 573.1261, Y 45.8901, Z -8.0000, A 0.000, B 0.000, C 0.000 }
gfCNCPoint6[12489] = {X 572.8303, Y 46.7355, Z -8.0000, A 0.000, B 0.000, C 0.000 }
gfCNCPoint6[12490] = {X 572.3538, Y 47.4940, Z -8.0000, A 0.000, B 0.000, C 0.000 }
gfCNCPoint6[12491] = {X 571.7204, Y 48.1273, Z -8.0000, A 0.000, B 0.000, C 0.000 }
gfCNCPoint6[12492] = {X 570.9620, Y 48.6039, Z -8.0000, A 0.000, B 0.000, C 0.000 }
gfCNCPoint6[12493] = {X 570.1165, Y 48.8997, Z -8.0000, A 0.000, B 0.000, C 0.000 }
gfCNCPoint6[12494] = {X 569.2264, Y 49.0000, Z -8.0000, A 0.000, B 0.000, C 0.000 }
gfCNCPoint6[12495] = {X 562.4443, Y 49.0000, Z -8.0000, A 0.000, B 0.000, C 0.000 }
gfCNCPoint6[12496] = {X 561.5542, Y 48.8997, Z -8.0000, A 0.000, B 0.000, C 0.000 }
gfCNCPoint6[12497] = {X 560.7088, Y 48.6039, Z -8.0000, A 0.000, B 0.000, C 0.000 }
gfCNCPoint6[12498] = {X 559.9503, Y 48.1273, Z -8.0000, A 0.000, B 0.000, C 0.000 }
gfCNCPoint6[12499] = {X 559.3170, Y 47.4940, Z -8.0000, A 0.000, B 0.000, C 0.000 }
gfCNCPoint6[12500] = {X 558.8404, Y 46.7355, Z -8.0000, A 0.000, B 0.000, C 0.000 }
gfCNCPoint6[12501] = {X 558.5446, Y 45.8901, Z -8.0000, A 0.000, B 0.000, C 0.000 }
gfCNCPoint6[12502] = {X 558.4443, Y 45.0000, Z -8.0000, A 0.000, B 0.000, C 0.000 }
gfCNCPoint6[12503] = {X 558.4443, Y 44.0660, Z -8.0000, A 0.000, B 0.000, C 0.000 }
gfCNCPoint6[12504] = {X 558.5382, Y 43.2136, Z -8.0000, A 0.000, B 0.000, C 0.000 }
gfCNCPoint6[12505] = {X 558.8104, Y 42.4005, Z -8.0000, A 0.000, B 0.000, C 0.000 }
gfCNCPoint6[12506] = {X 559.2485, Y 41.6634, Z -8.0000, A 0.000, B 0.000, C 0.000 }
gfCNCPoint6[12507] = {X 559.8327, Y 41.0357, Z -8.0000, A 0.000, B 0.000, C 0.000 }
gfCNCPoint6[12508] = {X 559.9010, Y 40.9778, Z -8.0000, A 0.000, B 0.000, C 0.000 }
gfCNCPoint6[12509] = {X 559.9706, Y 40.9214, Z -8.0000, A 0.000, B 0.000, C 0.000 }
gfCNCPoint6[12510] = {X 559.9710, Y 9.0778, Z -8.0000, A 0.000, B 0.000, C 0.000 }
gfCNCPoint6[12511] = {X 559.3293, Y 8.4435, Z -8.0000, A 0.000, B 0.000, C 0.000 }
gfCNCPoint6[12512] = {X 558.8462, Y 7.6814, Z -8.0000, A 0.000, B 0.000, C 0.000 }
gfCNCPoint6[12513] = {X 558.5460, Y 6.8305, Z -8.0000, A 0.000, B 0.000, C 0.000 }
gfCNCPoint6[12514] = {X 558.4443, Y 5.9340, Z -8.0000, A 0.000, B 0.000, C 0.000 }
gfCNCPoint6[12515] = {X 558.4443, Y 5.0000, Z -8.0000, A 0.000, B 0.000, C 0.000 }
gfCNCPoint6[12516] = {X 558.5446, Y 4.1099, Z -8.0000, A 0.000, B 0.000, C 0.000 }
gfCNCPoint6[12517] = {X 558.8404, Y 3.2645, Z -8.0000, A 0.000, B 0.000, C 0.000 }
gfCNCPoint6[12518] = {X 559.3170, Y 2.5060, Z -8.0000, A 0.000, B 0.000, C 0.000 }
gfCNCPoint6[12519] = {X 559.9503, Y 1.8727, Z -8.0000, A 0.000, B 0.000, C 0.000 }
gfCNCPoint6[12520] = {X 560.7088, Y 1.3961, Z -8.0000, A 0.000, B 0.000, C 0.000 }
gfCNCPoint6[12521] = {X 561.5542, Y 1.1003, Z -8.0000, A 0.000, B 0.000, C 0.000 }
gfCNCPoint6[12522] = {X 562.4443, Y 1.0000, Z -8.0000, A 0.000, B 0.000, C 0.000 }
gfCNCPoint6[12523] = {X 570.9376, Y 1.0000, Z -8.0000, A 0.000, B 0.000, C 0.000 }
gfCNCPoint6[12524] = {X 571.8276, Y 1.1003, Z -8.0000, A 0.000, B 0.000, C 0.000 }
gfCNCPoint6[12525] = {X 572.6731, Y 1.3961, Z -8.0000, A 0.000, B 0.000, C 0.000 }
gfCNCPoint6[12526] = {X 573.4315, Y 1.8727, Z -8.0000, A 0.000, B 0.000, C 0.000 }
gfCNCPoint6[12527] = {X 574.0649, Y 2.5060, Z -8.0000, A 0.000, B 0.000, C 0.000 }
gfCNCPoint6[12528] = {X 574.5414, Y 3.2645, Z -8.0000, A 0.000, B 0.000, C 0.000 }
gfCNCPoint6[12529] = {X 574.8373, Y 4.1099, Z -8.0000, A 0.000, B 0.000, C 0.000 }
gfCNCPoint6[12530] = {X 574.9376, Y 5.0000, Z -8.0000, A 0.000, B 0.000, C 0.000 }
gfCNCPoint6[12531] = {X 574.9372, Y 5.9858, Z -8.0000, A 0.000, B 0.000, C 0.000 }
gfCNCPoint6[12532] = {X 574.8650, Y 6.6924, Z -8.0000, A 0.000, B 0.000, C 0.000 }
gfCNCPoint6[12533] = {X 574.6690, Y 7.3751, Z -8.0000, A 0.000, B 0.000, C 0.000 }
gfCNCPoint6[12534] = {X 574.3553, Y 8.0123, Z -8.0000, A 0.000, B 0.000, C 0.000 }
gfCNCPoint6[12535] = {X 574.2923, Y 8.1125, Z -8.0000, A 0.000, B 0.000, C 0.000 }
gfCNCPoint6[12536] = {X 574.2264, Y 8.2108, Z -8.0000, A 0.000, B 0.000, C 0.000 }
gfCNCPoint6[12537] = {X 574.2622, Y 8.2359, Z -8.0000, A 0.000, B 0.000, C 0.000 }
gfCNCPoint6[12538] = {X 574.2861, Y 8.2725, Z -8.0000, A 0.000, B 0.000, C 0.000 }
gfCNCPoint6[12539] = {X 574.9161, Y 9.8064, Z -8.0000, A 0.000, B 0.000, C 0.000 }
gfCNCPoint6[12540] = {X 581.1904, Y 25.2153, Z -8.0000, A 0.000, B 0.000, C 0.000 }
gfCNCPoint6[12541] = {X 588.2024, Y 8.0660, Z -8.0000, A 0.000, B 0.000, C 0.000 }
gfCNCPoint6[12542] = {X 588.1527, Y 7.9848, Z -8.0000, A 0.000, B 0.000, C 0.000 }
gfCNCPoint6[12543] = {X 588.1048, Y 7.9025, Z -8.0000, A 0.000, B 0.000, C 0.000 }
gfCNCPoint6[12544] = {X 587.8200, Y 7.2794, Z -8.0000, A 0.000, B 0.000, C 0.000 }
gfCNCPoint6[12545] = {X 587.6456, Y 6.6167, Z -8.0000, A 0.000, B 0.000, C 0.000 }
gfCNCPoint6[12546] = {X 587.5870, Y 5.9340, Z -8.0000, A 0.000, B 0.000, C 0.000 }
gfCNCPoint6[12547] = {X 587.5870, Y 5.0000, Z -8.0000, A 0.000, B 0.000, C 0.000 }
gfCNCPoint6[12548] = {X 587.6872, Y 4.1099, Z -8.0000, A 0.000, B 0.000, C 0.000 }
gfCNCPoint6[12549] = {X 587.9831, Y 3.2645, Z -8.0000, A 0.000, B 0.000, C 0.000 }
gfCNCPoint6[12550] = {X 588.4596, Y 2.5060, Z -8.0000, A 0.000, B 0.000, C 0.000 }
gfCNCPoint6[12551] = {X 589.0930, Y 1.8727, Z -8.0000, A 0.000, B 0.000, C 0.000 }
gfCNCPoint6[12552] = {X 589.8514, Y 1.3961, Z -8.0000, A 0.000, B 0.000, C 0.000 }
gfCNCPoint6[12553] = {X 590.6969, Y 1.1003, Z -8.0000, A 0.000, B 0.000, C 0.000 }
gfCNCPoint6[12554] = {X 591.5870, Y 1.0000, Z -8.0000, A 0.000, B 0.000, C 0.000 }
gfCNCPoint6[12555] = {X 600.0000, Y 1.0000, Z -8.0000, A 0.000, B 0.000, C 0.000 }
gfCNCPoint6[12556] = {X 600.7928, Y 1.0793, Z -8.0000, A 0.000, B 0.000, C 0.000 }
gfCNCPoint6[12557] = {X 601.5541, Y 1.3142, Z -8.0000, A 0.000, B 0.000, C 0.000 }
gfCNCPoint6[12558] = {X 602.2538, Y 1.6954, Z -8.0000, A 0.000, B 0.000, C 0.000 }
gfCNCPoint6[12559] = {X 602.8640, Y 2.2076, Z -8.0000, A 0.000, B 0.000, C 0.000 }
gfCNCPoint6[12560] = {X 603.3606, Y 2.8306, Z -8.0000, A 0.000, B 0.000, C 0.000 }
gfCNCPoint6[12561] = {X 603.5432, Y 3.1438, Z -8.0000, A 0.000, B 0.000, C 0.000 }
gfCNCPoint6[12562] = {X 603.6967, Y 3.4721, Z -8.0000, A 0.000, B 0.000, C 0.000 }
gfCNCPoint6[12563] = {X 607.6967, Y 13.1500, Z -8.0000, A 0.000, B 0.000, C 0.000 }
gfCNCPoint6[12564] = {X 607.6967, Y 13.1500, Z -5.0000, A 0.000, B 0.000, C 0.000 }
gfCNCPoint6[12565] = {X 607.6967, Y 13.1500, Z 11.0000, A 0.000, B 0.000, C 0.000 }
gfCNCPoint6[12566] = {X 256.2481, Y 19.7827, Z 11.0000, A 0.000, B 0.000, C 0.000 }
gfCNCPoint6[12567] = {X 256.2481, Y 19.7827, Z -4.1667, A 0.000, B 0.000, C 0.000 }
gfCNCPoint6[12568] = {X 251.5292, Y 19.7824, Z -5.4311, A 0.000, B 0.000, C 0.000 }
gfCNCPoint6[12569] = {X 250.8342, Y 19.7932, Z -5.6173, A 0.000, B 0.000, C 0.000 }
gfCNCPoint6[12570] = {X 250.1827, Y 19.7941, Z -5.7919, A 0.000, B 0.000, C 0.000 }
gfCNCPoint6[12571] = {X 249.4936, Y 19.8930, Z -5.9784, A 0.000, B 0.000, C 0.000 }
gfCNCPoint6[12572] = {X 248.8455, Y 20.0813, Z -6.1593, A 0.000, B 0.000, C 0.000 }
gfCNCPoint6[12573] = {X 248.7088, Y 20.1126, Z -6.1969, A 0.000, B 0.000, C 0.000 }
gfCNCPoint6[12574] = {X 248.6554, Y 20.1627, Z -6.2165, A 0.000, B 0.000, C 0.000 }
gfCNCPoint6[12575] = {X 248.6155, Y 20.2971, Z -6.2540, A 0.000, B 0.000, C 0.000 }
gfCNCPoint6[12576] = {X 248.4765, Y 20.7655, Z -6.3850, A 0.000, B 0.000, C 0.000 }
gfCNCPoint6[12577] = {X 248.4463, Y 21.8662, Z -6.6800, A 0.000, B 0.000, C 0.000 }
gfCNCPoint6[12578] = {X 248.5594, Y 22.3415, Z -6.8109, A 0.000, B 0.000, C 0.000 }
gfCNCPoint6[12579] = {X 248.8774, Y 22.4370, Z -6.8999, A 0.000, B 0.000, C 0.000 }
gfCNCPoint6[12580] = {X 249.2083, Y 22.4639, Z -6.9889, A 0.000, B 0.000, C 0.000 }
gfCNCPoint6[12581] = {X 250.4445, Y 22.5643, Z -7.3212, A 0.000, B 0.000, C 0.000 }
gfCNCPoint6[12582] = {X 251.6873, Y 22.5560, Z -7.6542, A 0.000, B 0.000, C 0.000 }
gfCNCPoint6[12583] = {X 252.9779, Y 22.5560, Z -8.0000, A 0.000, B 0.000, C 0.000 }
gfCNCPoint6[12584] = {X 257.4115, Y 22.5560, Z -8.0000, A 0.000, B 0.000, C 0.000 }
gfCNCPoint6[12585] = {X 257.4115, Y 19.7828, Z -8.0000, A 0.000, B 0.000, C 0.000 }
gfCNCPoint6[12586] = {X 251.5292, Y 19.7824, Z -8.0000, A 0.000, B 0.000, C 0.000 }
gfCNCPoint6[12587] = {X 250.8342, Y 19.7932, Z -8.0000, A 0.000, B 0.000, C 0.000 }
gfCNCPoint6[12588] = {X 249.8295, Y 19.8661, Z -8.0000, A 0.000, B 0.000, C 0.000 }
gfCNCPoint6[12589] = {X 248.8455, Y 20.0813, Z -8.0000, A 0.000, B 0.000, C 0.000 }
gfCNCPoint6[12590] = {X 248.7013, Y 20.1581, Z -8.0000, A 0.000, B 0.000, C 0.000 }
gfCNCPoint6[12591] = {X 248.6155, Y 20.2971, Z -8.0000, A 0.000, B 0.000, C 0.000 }
gfCNCPoint6[12592] = {X 248.4777, Y 20.9718, Z -8.0000, A 0.000, B 0.000, C 0.000 }
gfCNCPoint6[12593] = {X 248.4588, Y 21.6602, Z -8.0000, A 0.000, B 0.000, C 0.000 }
gfCNCPoint6[12594] = {X 248.5594, Y 22.3415, Z -8.0000, A 0.000, B 0.000, C 0.000 }
gfCNCPoint6[12595] = {X 248.8806, Y 22.4198, Z -8.0000, A 0.000, B 0.000, C 0.000 }
gfCNCPoint6[12596] = {X 249.2083, Y 22.4639, Z -8.0000, A 0.000, B 0.000, C 0.000 }
gfCNCPoint6[12597] = {X 250.4468, Y 22.5372, Z -8.0000, A 0.000, B 0.000, C 0.000 }
gfCNCPoint6[12598] = {X 251.6873, Y 22.5560, Z -8.0000, A 0.000, B 0.000, C 0.000 }
gfCNCPoint6[12599] = {X 252.9779, Y 22.5560, Z -8.0000, A 0.000, B 0.000, C 0.000 }
gfCNCPoint6[12600] = {X 248.9931, Y 22.2874, Z -8.0000, A 0.000, B 0.000, C 0.000 }
gfCNCPoint6[12601] = {X 252.9779, Y 22.6360, Z -8.0000, A 0.000, B 0.000, C 0.000 }
gfCNCPoint6[12602] = {X 257.4915, Y 22.6360, Z -8.0000, A 0.000, B 0.000, C 0.000 }
gfCNCPoint6[12603] = {X 257.4915, Y 19.7028, Z -8.0000, A 0.000, B 0.000, C 0.000 }
gfCNCPoint6[12604] = {X 251.5286, Y 19.7024, Z -8.0000, A 0.000, B 0.000, C 0.000 }
gfCNCPoint6[12605] = {X 250.8363, Y 19.7132, Z -8.0000, A 0.000, B 0.000, C 0.000 }
gfCNCPoint6[12606] = {X 249.8258, Y 19.7862, Z -8.0000, A 0.000, B 0.000, C 0.000 }
gfCNCPoint6[12607] = {X 248.8358, Y 20.0015, Z -8.0000, A 0.000, B 0.000, C 0.000 }
gfCNCPoint6[12608] = {X 248.6496, Y 20.0969, Z -8.0000, A 0.000, B 0.000, C 0.000 }
gfCNCPoint6[12609] = {X 248.5388, Y 20.2743, Z -8.0000, A 0.000, B 0.000, C 0.000 }
gfCNCPoint6[12610] = {X 248.3965, Y 20.9779, Z -8.0000, A 0.000, B 0.000, C 0.000 }
gfCNCPoint6[12611] = {X 248.3809, Y 21.6955, Z -8.0000, A 0.000, B 0.000, C 0.000 }
gfCNCPoint6[12612] = {X 248.4924, Y 22.4046, Z -8.0000, A 0.000, B 0.000, C 0.000 }
gfCNCPoint6[12613] = {X 248.8432, Y 22.4941, Z -8.0000, A 0.000, B 0.000, C 0.000 }
gfCNCPoint6[12614] = {X 249.2019, Y 22.5436, Z -8.0000, A 0.000, B 0.000, C 0.000 }
gfCNCPoint6[12615] = {X 250.4431, Y 22.6171, Z -8.0000, A 0.000, B 0.000, C 0.000 }
gfCNCPoint6[12616] = {X 251.6863, Y 22.6360, Z -8.0000, A 0.000, B 0.000, C 0.000 }
gfCNCPoint6[12617] = {X 252.9779, Y 22.6360, Z -8.0000, A 0.000, B 0.000, C 0.000 }
gfCNCPoint6[12618] = {X 256.9627, Y 22.2874, Z -8.0000, A 0.000, B 0.000, C 0.000 }
gfCNCPoint6[12619] = {X 248.9931, Y 22.3674, Z -8.0000, A 0.000, B 0.000, C 0.000 }
gfCNCPoint6[12620] = {X 252.9779, Y 22.7160, Z -8.0000, A 0.000, B 0.000, C 0.000 }
gfCNCPoint6[12621] = {X 257.5715, Y 22.7160, Z -8.0000, A 0.000, B 0.000, C 0.000 }
gfCNCPoint6[12622] = {X 257.5715, Y 19.6228, Z -8.0000, A 0.000, B 0.000, C 0.000 }
gfCNCPoint6[12623] = {X 251.5280, Y 19.6224, Z -8.0000, A 0.000, B 0.000, C 0.000 }
gfCNCPoint6[12624] = {X 250.8357, Y 19.6332, Z -8.0000, A 0.000, B 0.000, C 0.000 }
gfCNCPoint6[12625] = {X 249.8156, Y 19.7069, Z -8.0000, A 0.000, B 0.000, C 0.000 }
gfCNCPoint6[12626] = {X 248.8162, Y 19.9239, Z -8.0000, A 0.000, B 0.000, C 0.000 }
gfCNCPoint6[12627] = {X 248.5942, Y 20.0392, Z -8.0000, A 0.000, B 0.000, C 0.000 }
gfCNCPoint6[12628] = {X 248.4621, Y 20.2516, Z -8.0000, A 0.000, B 0.000, C 0.000 }
gfCNCPoint6[12629] = {X 248.3154, Y 20.9838, Z -8.0000, A 0.000, B 0.000, C 0.000 }
gfCNCPoint6[12630] = {X 248.3032, Y 21.7305, Z -8.0000, A 0.000, B 0.000, C 0.000 }
gfCNCPoint6[12631] = {X 248.4259, Y 22.4671, Z -8.0000, A 0.000, B 0.000, C 0.000 }
gfCNCPoint6[12632] = {X 248.8060, Y 22.5682, Z -8.0000, A 0.000, B 0.000, C 0.000 }
gfCNCPoint6[12633] = {X 249.1954, Y 22.6234, Z -8.0000, A 0.000, B 0.000, C 0.000 }
gfCNCPoint6[12634] = {X 250.4400, Y 22.6970, Z -8.0000, A 0.000, B 0.000, C 0.000 }
gfCNCPoint6[12635] = {X 251.6865, Y 22.7160, Z -8.0000, A 0.000, B 0.000, C 0.000 }
gfCNCPoint6[12636] = {X 252.9779, Y 22.7160, Z -8.0000, A 0.000, B 0.000, C 0.000 }
gfCNCPoint6[12637] = {X 256.9627, Y 22.3674, Z -8.0000, A 0.000, B 0.000, C 0.000 }
gfCNCPoint6[12638] = {X 248.9931, Y 22.4474, Z -8.0000, A 0.000, B 0.000, C 0.000 }
gfCNCPoint6[12639] = {X 252.9779, Y 22.7960, Z -8.0000, A 0.000, B 0.000, C 0.000 }
gfCNCPoint6[12640] = {X 257.6515, Y 22.7960, Z -8.0000, A 0.000, B 0.000, C 0.000 }
gfCNCPoint6[12641] = {X 257.6515, Y 19.5428, Z -8.0000, A 0.000, B 0.000, C 0.000 }
gfCNCPoint6[12642] = {X 251.5274, Y 19.5424, Z -8.0000, A 0.000, B 0.000, C 0.000 }
gfCNCPoint6[12643] = {X 250.8350, Y 19.5532, Z -8.0000, A 0.000, B 0.000, C 0.000 }
gfCNCPoint6[12644] = {X 249.8053, Y 19.6275, Z -8.0000, A 0.000, B 0.000, C 0.000 }
gfCNCPoint6[12645] = {X 248.7963, Y 19.8463, Z -8.0000, A 0.000, B 0.000, C 0.000 }
gfCNCPoint6[12646] = {X 248.5387, Y 19.9815, Z -8.0000, A 0.000, B 0.000, C 0.000 }
gfCNCPoint6[12647] = {X 248.3854, Y 20.2288, Z -8.0000, A 0.000, B 0.000, C 0.000 }
gfCNCPoint6[12648] = {X 248.2344, Y 20.9896, Z -8.0000, A 0.000, B 0.000, C 0.000 }
gfCNCPoint6[12649] = {X 248.2256, Y 21.7652, Z -8.0000, A 0.000, B 0.000, C 0.000 }
gfCNCPoint6[12650] = {X 248.3596, Y 22.5292, Z -8.0000, A 0.000, B 0.000, C 0.000 }
gfCNCPoint6[12651] = {X 248.7688, Y 22.6422, Z -8.0000, A 0.000, B 0.000, C 0.000 }
gfCNCPoint6[12652] = {X 249.1890, Y 22.7031, Z -8.0000, A 0.000, B 0.000, C 0.000 }
gfCNCPoint6[12653] = {X 250.4369, Y 22.7770, Z -8.0000, A 0.000, B 0.000, C 0.000 }
gfCNCPoint6[12654] = {X 251.6868, Y 22.7960, Z -8.0000, A 0.000, B 0.000, C 0.000 }
gfCNCPoint6[12655] = {X 252.9779, Y 22.7960, Z -8.0000, A 0.000, B 0.000, C 0.000 }
gfCNCPoint6[12656] = {X 256.9627, Y 22.4474, Z -8.0000, A 0.000, B 0.000, C 0.000 }
gfCNCPoint6[12657] = {X 248.9931, Y 22.5274, Z -8.0000, A 0.000, B 0.000, C 0.000 }
gfCNCPoint6[12658] = {X 252.9779, Y 22.8760, Z -8.0000, A 0.000, B 0.000, C 0.000 }
gfCNCPoint6[12659] = {X 257.7315, Y 22.8760, Z -8.0000, A 0.000, B 0.000, C 0.000 }
gfCNCPoint6[12660] = {X 257.7315, Y 19.4628, Z -8.0000, A 0.000, B 0.000, C 0.000 }
gfCNCPoint6[12661] = {X 251.5267, Y 19.4624, Z -8.0000, A 0.000, B 0.000, C 0.000 }
gfCNCPoint6[12662] = {X 250.8343, Y 19.4732, Z -8.0000, A 0.000, B 0.000, C 0.000 }
gfCNCPoint6[12663] = {X 249.7949, Y 19.5482, Z -8.0000, A 0.000, B 0.000, C 0.000 }
gfCNCPoint6[12664] = {X 248.7763, Y 19.7688, Z -8.0000, A 0.000, B 0.000, C 0.000 }
gfCNCPoint6[12665] = {X 248.4831, Y 19.9240, Z -8.0000, A 0.000, B 0.000, C 0.000 }
gfCNCPoint6[12666] = {X 248.3087, Y 20.2061, Z -8.0000, A 0.000, B 0.000, C 0.000 }
gfCNCPoint6[12667] = {X 248.1540, Y 20.9889, Z -8.0000, A 0.000, B 0.000, C 0.000 }
gfCNCPoint6[12668] = {X 248.1472, Y 21.7869, Z -8.0000, A 0.000, B 0.000, C 0.000 }
gfCNCPoint6[12669] = {X 248.2885, Y 22.5722, Z -8.0000, A 0.000, B 0.000, C 0.000 }
gfCNCPoint6[12670] = {X 248.3072, Y 22.5956, Z -8.0000, A 0.000, B 0.000, C 0.000 }
gfCNCPoint6[12671] = {X 248.3335, Y 22.6048, Z -8.0000, A 0.000, B 0.000, C 0.000 }
gfCNCPoint6[12672] = {X 248.7524, Y 22.7205, Z -8.0000, A 0.000, B 0.000, C 0.000 }
gfCNCPoint6[12673] = {X 249.1825, Y 22.7828, Z -8.0000, A 0.000, B 0.000, C 0.000 }
gfCNCPoint6[12674] = {X 250.4338, Y 22.8569, Z -8.0000, A 0.000, B 0.000, C 0.000 }
gfCNCPoint6[12675] = {X 251.6871, Y 22.8760, Z -8.0000, A 0.000, B 0.000, C 0.000 }
gfCNCPoint6[12676] = {X 252.9779, Y 22.8760, Z -8.0000, A 0.000, B 0.000, C 0.000 }
gfCNCPoint6[12677] = {X 256.9627, Y 22.5274, Z -8.0000, A 0.000, B 0.000, C 0.000 }
gfCNCPoint6[12678] = {X 252.9779, Y 20.9560, Z -8.0000, A 0.000, B 0.000, C 0.000 }
gfCNCPoint6[12679] = {X 252.9779, Y 22.9560, Z -8.0000, A 0.000, B 0.000, C 0.000 }
gfCNCPoint6[12680] = {X 257.8115, Y 22.9560, Z -8.0000, A 0.000, B 0.000, C 0.000 }
gfCNCPoint6[12681] = {X 257.8115, Y 19.3828, Z -8.0000, A 0.000, B 0.000, C 0.000 }
gfCNCPoint6[12682] = {X 251.5261, Y 19.3824, Z -8.0000, A 0.000, B 0.000, C 0.000 }
gfCNCPoint6[12683] = {X 250.8336, Y 19.3932, Z -8.0000, A 0.000, B 0.000, C 0.000 }
gfCNCPoint6[12684] = {X 249.7844, Y 19.4689, Z -8.0000, A 0.000, B 0.000, C 0.000 }
gfCNCPoint6[12685] = {X 248.7562, Y 19.6914, Z -8.0000, A 0.000, B 0.000, C 0.000 }
gfCNCPoint6[12686] = {X 248.4275, Y 19.8664, Z -8.0000, A 0.000, B 0.000, C 0.000 }
gfCNCPoint6[12687] = {X 248.2320, Y 20.1833, Z -8.0000, A 0.000, B 0.000, C 0.000 }
gfCNCPoint6[12688] = {X 248.0739, Y 20.9862, Z -8.0000, A 0.000, B 0.000, C 0.000 }
gfCNCPoint6[12689] = {X 248.0684, Y 21.8045, Z -8.0000, A 0.000, B 0.000, C 0.000 }
gfCNCPoint6[12690] = {X 248.2158, Y 22.6095, Z -8.0000, A 0.000, B 0.000, C 0.000 }
gfCNCPoint6[12691] = {X 248.2588, Y 22.6633, Z -8.0000, A 0.000, B 0.000, C 0.000 }
gfCNCPoint6[12692] = {X 248.7108, Y 22.7935, Z -8.0000, A 0.000, B 0.000, C 0.000 }
gfCNCPoint6[12693] = {X 249.1760, Y 22.8626, Z -8.0000, A 0.000, B 0.000, C 0.000 }
gfCNCPoint6[12694] = {X 250.4306, Y 22.9368, Z -8.0000, A 0.000, B 0.000, C 0.000 }
gfCNCPoint6[12695] = {X 251.6873, Y 22.9560, Z -8.0000, A 0.000, B 0.000, C 0.000 }
gfCNCPoint6[12696] = {X 252.9779, Y 22.9560, Z -8.0000, A 0.000, B 0.000, C 0.000 }
gfCNCPoint6[12697] = {X 256.9627, Y 22.6074, Z -8.0000, A 0.000, B 0.000, C 0.000 }
gfCNCPoint6[12698] = {X 256.9627, Y 22.6074, Z -5.0000, A 0.000, B 0.000, C 0.000 }
gfCNCPoint6[12699] = {X 256.9627, Y 22.6074, Z 11.0000, A 0.000, B 0.000, C 0.000 }
gfCNCPoint6[12700] = {X 188.5005, Y 19.4692, Z 11.0000, A 0.000, B 0.000, C 0.000 }
gfCNCPoint6[12701] = {X 188.5005, Y 19.4692, Z -4.1667, A 0.000, B 0.000, C 0.000 }
gfCNCPoint6[12702] = {X 188.3879, Y 19.4294, Z -4.1987, A 0.000, B 0.000, C 0.000 }
gfCNCPoint6[12703] = {X 187.7714, Y 19.3612, Z -4.3649, A 0.000, B 0.000, C 0.000 }
gfCNCPoint6[12704] = {X 186.9109, Y 19.2613, Z -4.5970, A 0.000, B 0.000, C 0.000 }
gfCNCPoint6[12705] = {X 184.5930, Y 19.3688, Z -5.2187, A 0.000, B 0.000, C 0.000 }
gfCNCPoint6[12706] = {X 183.7426, Y 19.5485, Z -5.4516, A 0.000, B 0.000, C 0.000 }
gfCNCPoint6[12707] = {X 183.0434, Y 19.6910, Z -5.6428, A 0.000, B 0.000, C 0.000 }
gfCNCPoint6[12708] = {X 182.0225, Y 20.0626, Z -5.9339, A 0.000, B 0.000, C 0.000 }
gfCNCPoint6[12709] = {X 181.3953, Y 20.4028, Z -6.1251, A 0.000, B 0.000, C 0.000 }
gfCNCPoint6[12710] = {X 181.3392, Y 20.9144, Z -6.2630, A 0.000, B 0.000, C 0.000 }
gfCNCPoint6[12711] = {X 180.8657, Y 22.1248, Z -6.6113, A 0.000, B 0.000, C 0.000 }
gfCNCPoint6[12712] = {X 180.5597, Y 22.5387, Z -6.7492, A 0.000, B 0.000, C 0.000 }
gfCNCPoint6[12713] = {X 182.2924, Y 22.3328, Z -7.2168, A 0.000, B 0.000, C 0.000 }
gfCNCPoint6[12714] = {X 182.5945, Y 22.3083, Z -7.2980, A 0.000, B 0.000, C 0.000 }
gfCNCPoint6[12715] = {X 184.3413, Y 22.2321, Z -7.7665, A 0.000, B 0.000, C 0.000 }
gfCNCPoint6[12716] = {X 184.7768, Y 22.2170, Z -7.8832, A 0.000, B 0.000, C 0.000 }
gfCNCPoint6[12717] = {X 185.2122, Y 22.1986, Z -8.0000, A 0.000, B 0.000, C 0.000 }
gfCNCPoint6[12718] = {X 187.5422, Y 22.0762, Z -8.0000, A 0.000, B 0.000, C 0.000 }
gfCNCPoint6[12719] = {X 189.8692, Y 21.9067, Z -8.0000, A 0.000, B 0.000, C 0.000 }
gfCNCPoint6[12720] = {X 190.4705, Y 21.8298, Z -8.0000, A 0.000, B 0.000, C 0.000 }
gfCNCPoint6[12721] = {X 191.0576, Y 21.6787, Z -8.0000, A 0.000, B 0.000, C 0.000 }
gfCNCPoint6[12722] = {X 191.0672, Y 21.1640, Z -8.0000, A 0.000, B 0.000, C 0.000 }
gfCNCPoint6[12723] = {X 190.8720, Y 20.6877, Z -8.0000, A 0.000, B 0.000, C 0.000 }
gfCNCPoint6[12724] = {X 190.5040, Y 20.3279, Z -8.0000, A 0.000, B 0.000, C 0.000 }
gfCNCPoint6[12725] = {X 189.6464, Y 19.8666, Z -8.0000, A 0.000, B 0.000, C 0.000 }
gfCNCPoint6[12726] = {X 188.7283, Y 19.5418, Z -8.0000, A 0.000, B 0.000, C 0.000 }
gfCNCPoint6[12727] = {X 187.7714, Y 19.3612, Z -8.0000, A 0.000, B 0.000, C 0.000 }
gfCNCPoint6[12728] = {X 186.4243, Y 19.2781, Z -8.0000, A 0.000, B 0.000, C 0.000 }
gfCNCPoint6[12729] = {X 185.0761, Y 19.3408, Z -8.0000, A 0.000, B 0.000, C 0.000 }
gfCNCPoint6[12730] = {X 183.7426, Y 19.5485, Z -8.0000, A 0.000, B 0.000, C 0.000 }
gfCNCPoint6[12731] = {X 182.5373, Y 19.8887, Z -8.0000, A 0.000, B 0.000, C 0.000 }
gfCNCPoint6[12732] = {X 181.3953, Y 20.4028, Z -8.0000, A 0.000, B 0.000, C 0.000 }
gfCNCPoint6[12733] = {X 181.2440, Y 21.1603, Z -8.0000, A 0.000, B 0.000, C 0.000 }
gfCNCPoint6[12734] = {X 180.9626, Y 21.8797, Z -8.0000, A 0.000, B 0.000, C 0.000 }
gfCNCPoint6[12735] = {X 180.5597, Y 22.5387, Z -8.0000, A 0.000, B 0.000, C 0.000 }
gfCNCPoint6[12736] = {X 182.4476, Y 22.3501, Z -8.0000, A 0.000, B 0.000, C 0.000 }
gfCNCPoint6[12737] = {X 184.3413, Y 22.2321, Z -8.0000, A 0.000, B 0.000, C 0.000 }
gfCNCPoint6[12738] = {X 184.7768, Y 22.2162, Z -8.0000, A 0.000, B 0.000, C 0.000 }
gfCNCPoint6[12739] = {X 185.2122, Y 22.1986, Z -8.0000, A 0.000, B 0.000, C 0.000 }
gfCNCPoint6[12740] = {X 181.2196, Y 22.0988, Z -8.0000, A 0.000, B 0.000, C 0.000 }
gfCNCPoint6[12741] = {X 185.2156, Y 22.2785, Z -8.0000, A 0.000, B 0.000, C 0.000 }
gfCNCPoint6[12742] = {X 187.5450, Y 22.1562, Z -8.0000, A 0.000, B 0.000, C 0.000 }
gfCNCPoint6[12743] = {X 189.8715, Y 21.9867, Z -8.0000, A 0.000, B 0.000, C 0.000 }
gfCNCPoint6[12744] = {X 190.5061, Y 21.9044, Z -8.0000, A 0.000, B 0.000, C 0.000 }
gfCNCPoint6[12745] = {X 191.1248, Y 21.7407, Z -8.0000, A 0.000, B 0.000, C 0.000 }
gfCNCPoint6[12746] = {X 191.1511, Y 21.1793, Z -8.0000, A 0.000, B 0.000, C 0.000 }
gfCNCPoint6[12747] = {X 190.9468, Y 20.6557, Z -8.0000, A 0.000, B 0.000, C 0.000 }
gfCNCPoint6[12748] = {X 190.5472, Y 20.2605, Z -8.0000, A 0.000, B 0.000, C 0.000 }
gfCNCPoint6[12749] = {X 189.6795, Y 19.7937, Z -8.0000, A 0.000, B 0.000, C 0.000 }
gfCNCPoint6[12750] = {X 188.7506, Y 19.4650, Z -8.0000, A 0.000, B 0.000, C 0.000 }
gfCNCPoint6[12751] = {X 187.7824, Y 19.2820, Z -8.0000, A 0.000, B 0.000, C 0.000 }
gfCNCPoint6[12752] = {X 186.4271, Y 19.1981, Z -8.0000, A 0.000, B 0.000, C 0.000 }
gfCNCPoint6[12753] = {X 185.0707, Y 19.2609, Z -8.0000, A 0.000, B 0.000, C 0.000 }
gfCNCPoint6[12754] = {X 183.7289, Y 19.4697, Z -8.0000, A 0.000, B 0.000, C 0.000 }
gfCNCPoint6[12755] = {X 182.4919, Y 19.8201, Z -8.0000, A 0.000, B 0.000, C 0.000 }
gfCNCPoint6[12756] = {X 181.3215, Y 20.3519, Z -8.0000, A 0.000, B 0.000, C 0.000 }
gfCNCPoint6[12757] = {X 181.1582, Y 21.1712, Z -8.0000, A 0.000, B 0.000, C 0.000 }
gfCNCPoint6[12758] = {X 180.8404, Y 21.9437, Z -8.0000, A 0.000, B 0.000, C 0.000 }
gfCNCPoint6[12759] = {X 180.3797, Y 22.6406, Z -8.0000, A 0.000, B 0.000, C 0.000 }
gfCNCPoint6[12760] = {X 182.3580, Y 22.4375, Z -8.0000, A 0.000, B 0.000, C 0.000 }
gfCNCPoint6[12761] = {X 184.3427, Y 22.3121, Z -8.0000, A 0.000, B 0.000, C 0.000 }
gfCNCPoint6[12762] = {X 184.7792, Y 22.2961, Z -8.0000, A 0.000, B 0.000, C 0.000 }
gfCNCPoint6[12763] = {X 185.2156, Y 22.2785, Z -8.0000, A 0.000, B 0.000, C 0.000 }
gfCNCPoint6[12764] = {X 189.1821, Y 21.7615, Z -8.0000, A 0.000, B 0.000, C 0.000 }
gfCNCPoint6[12765] = {X 181.2230, Y 22.1788, Z -8.0000, A 0.000, B 0.000, C 0.000 }
gfCNCPoint6[12766] = {X 185.2190, Y 22.3584, Z -8.0000, A 0.000, B 0.000, C 0.000 }
gfCNCPoint6[12767] = {X 187.5497, Y 22.2360, Z -8.0000, A 0.000, B 0.000, C 0.000 }
gfCNCPoint6[12768] = {X 189.8774, Y 22.0665, Z -8.0000, A 0.000, B 0.000, C 0.000 }
gfCNCPoint6[12769] = {X 190.5428, Y 21.9787, Z -8.0000, A 0.000, B 0.000, C 0.000 }
gfCNCPoint6[12770] = {X 191.1905, Y 21.8029, Z -8.0000, A 0.000, B 0.000, C 0.000 }
gfCNCPoint6[12771] = {X 191.2481, Y 21.3479, Z -8.0000, A 0.000, B 0.000, C 0.000 }
gfCNCPoint6[12772] = {X 191.1588, Y 20.8980, Z -8.0000, A 0.000, B 0.000, C 0.000 }
gfCNCPoint6[12773] = {X 190.9318, Y 20.4995, Z -8.0000, A 0.000, B 0.000, C 0.000 }
gfCNCPoint6[12774] = {X 190.5904, Y 20.1932, Z -8.0000, A 0.000, B 0.000, C 0.000 }
gfCNCPoint6[12775] = {X 189.7119, Y 19.7206, Z -8.0000, A 0.000, B 0.000, C 0.000 }
gfCNCPoint6[12776] = {X 188.7714, Y 19.3877, Z -8.0000, A 0.000, B 0.000, C 0.000 }
gfCNCPoint6[12777] = {X 187.7912, Y 19.2025, Z -8.0000, A 0.000, B 0.000, C 0.000 }
gfCNCPoint6[12778] = {X 186.4274, Y 19.1181, Z -8.0000, A 0.000, B 0.000, C 0.000 }
gfCNCPoint6[12779] = {X 185.0625, Y 19.1814, Z -8.0000, A 0.000, B 0.000, C 0.000 }
gfCNCPoint6[12780] = {X 183.7123, Y 19.3914, Z -8.0000, A 0.000, B 0.000, C 0.000 }
gfCNCPoint6[12781] = {X 182.4465, Y 19.7515, Z -8.0000, A 0.000, B 0.000, C 0.000 }
gfCNCPoint6[12782] = {X 181.2502, Y 20.2999, Z -8.0000, A 0.000, B 0.000, C 0.000 }
gfCNCPoint6[12783] = {X 181.2397, Y 20.3534, Z -8.0000, A 0.000, B 0.000, C 0.000 }
gfCNCPoint6[12784] = {X 181.0587, Y 21.2188, Z -8.0000, A 0.000, B 0.000, C 0.000 }
gfCNCPoint6[12785] = {X 180.7022, Y 22.0279, Z -8.0000, A 0.000, B 0.000, C 0.000 }
gfCNCPoint6[12786] = {X 180.1857, Y 22.7454, Z -8.0000, A 0.000, B 0.000, C 0.000 }
gfCNCPoint6[12787] = {X 182.2621, Y 22.5258, Z -8.0000, A 0.000, B 0.000, C 0.000 }
gfCNCPoint6[12788] = {X 184.3458, Y 22.3921, Z -8.0000, A 0.000, B 0.000, C 0.000 }
gfCNCPoint6[12789] = {X 184.7824, Y 22.3761, Z -8.0000, A 0.000, B 0.000, C 0.000 }
gfCNCPoint6[12790] = {X 185.2190, Y 22.3584, Z -8.0000, A 0.000, B 0.000, C 0.000 }
gfCNCPoint6[12791] = {X 189.1854, Y 21.8414, Z -8.0000, A 0.000, B 0.000, C 0.000 }
gfCNCPoint6[12792] = {X 181.2264, Y 22.2587, Z -8.0000, A 0.000, B 0.000, C 0.000 }
gfCNCPoint6[12793] = {X 185.2224, Y 22.4383, Z -8.0000, A 0.000, B 0.000, C 0.000 }
gfCNCPoint6[12794] = {X 187.5543, Y 22.3159, Z -8.0000, A 0.000, B 0.000, C 0.000 }
gfCNCPoint6[12795] = {X 189.8833, Y 22.1463, Z -8.0000, A 0.000, B 0.000, C 0.000 }
gfCNCPoint6[12796] = {X 190.5788, Y 22.0530, Z -8.0000, A 0.000, B 0.000, C 0.000 }
gfCNCPoint6[12797] = {X 191.2549, Y 21.8651, Z -8.0000, A 0.000, B 0.000, C 0.000 }
gfCNCPoint6[12798] = {X 191.3288, Y 21.3761, Z -8.0000, A 0.000, B 0.000, C 0.000 }
gfCNCPoint6[12799] = {X 191.2408, Y 20.8895, Z -8.0000, A 0.000, B 0.000, C 0.000 }
gfCNCPoint6[12800] = {X 191.0005, Y 20.4573, Z -8.0000, A 0.000, B 0.000, C 0.000 }
gfCNCPoint6[12801] = {X 190.6336, Y 20.1259, Z -8.0000, A 0.000, B 0.000, C 0.000 }
gfCNCPoint6[12802] = {X 189.7442, Y 19.6474, Z -8.0000, A 0.000, B 0.000, C 0.000 }
gfCNCPoint6[12803] = {X 188.7923, Y 19.3105, Z -8.0000, A 0.000, B 0.000, C 0.000 }
gfCNCPoint6[12804] = {X 187.8000, Y 19.1229, Z -8.0000, A 0.000, B 0.000, C 0.000 }
gfCNCPoint6[12805] = {X 186.4277, Y 19.0381, Z -8.0000, A 0.000, B 0.000, C 0.000 }
gfCNCPoint6[12806] = {X 185.0543, Y 19.1018, Z -8.0000, A 0.000, B 0.000, C 0.000 }
gfCNCPoint6[12807] = {X 183.6958, Y 19.3131, Z -8.0000, A 0.000, B 0.000, C 0.000 }
gfCNCPoint6[12808] = {X 182.4010, Y 19.6830, Z -8.0000, A 0.000, B 0.000, C 0.000 }
gfCNCPoint6[12809] = {X 181.1788, Y 20.2481, Z -8.0000, A 0.000, B 0.000, C 0.000 }
gfCNCPoint6[12810] = {X 181.1605, Y 20.3417, Z -8.0000, A 0.000, B 0.000, C 0.000 }
gfCNCPoint6[12811] = {X 180.9651, Y 21.2476, Z -8.0000, A 0.000, B 0.000, C 0.000 }
gfCNCPoint6[12812] = {X 180.5740, Y 22.0877, Z -8.0000, A 0.000, B 0.000, C 0.000 }
gfCNCPoint6[12813] = {X 180.0066, Y 22.8205, Z -8.0000, A 0.000, B 0.000, C 0.000 }
gfCNCPoint6[12814] = {X 180.1924, Y 22.8257, Z -8.0000, A 0.000, B 0.000, C 0.000 }
gfCNCPoint6[12815] = {X 182.2670, Y 22.6059, Z -8.0000, A 0.000, B 0.000, C 0.000 }
gfCNCPoint6[12816] = {X 184.3489, Y 22.4720, Z -8.0000, A 0.000, B 0.000, C 0.000 }
gfCNCPoint6[12817] = {X 184.7857, Y 22.4560, Z -8.0000, A 0.000, B 0.000, C 0.000 }
gfCNCPoint6[12818] = {X 185.2224, Y 22.4383, Z -8.0000, A 0.000, B 0.000, C 0.000 }
gfCNCPoint6[12819] = {X 189.1888, Y 21.9214, Z -8.0000, A 0.000, B 0.000, C 0.000 }
gfCNCPoint6[12820] = {X 181.2298, Y 22.3386, Z -8.0000, A 0.000, B 0.000, C 0.000 }
gfCNCPoint6[12821] = {X 185.2258, Y 22.5183, Z -8.0000, A 0.000, B 0.000, C 0.000 }
gfCNCPoint6[12822] = {X 187.5589, Y 22.3958, Z -8.0000, A 0.000, B 0.000, C 0.000 }
gfCNCPoint6[12823] = {X 189.8892, Y 22.2261, Z -8.0000, A 0.000, B 0.000, C 0.000 }
gfCNCPoint6[12824] = {X 190.6143, Y 22.1274, Z -8.0000, A 0.000, B 0.000, C 0.000 }
gfCNCPoint6[12825] = {X 191.3183, Y 21.9274, Z -8.0000, A 0.000, B 0.000, C 0.000 }
gfCNCPoint6[12826] = {X 191.4089, Y 21.4047, Z -8.0000, A 0.000, B 0.000, C 0.000 }
gfCNCPoint6[12827] = {X 191.3227, Y 20.8813, Z -8.0000, A 0.000, B 0.000, C 0.000 }
gfCNCPoint6[12828] = {X 191.0693, Y 20.4153, Z -8.0000, A 0.000, B 0.000, C 0.000 }
gfCNCPoint6[12829] = {X 190.6767, Y 20.0585, Z -8.0000, A 0.000, B 0.000, C 0.000 }
gfCNCPoint6[12830] = {X 189.7766, Y 19.5743, Z -8.0000, A 0.000, B 0.000, C 0.000 }
gfCNCPoint6[12831] = {X 188.8131, Y 19.2332, Z -8.0000, A 0.000, B 0.000, C 0.000 }
gfCNCPoint6[12832] = {X 187.8088, Y 19.0434, Z -8.0000, A 0.000, B 0.000, C 0.000 }
gfCNCPoint6[12833] = {X 186.4281, Y 18.9581, Z -8.0000, A 0.000, B 0.000, C 0.000 }
gfCNCPoint6[12834] = {X 185.0462, Y 19.0222, Z -8.0000, A 0.000, B 0.000, C 0.000 }
gfCNCPoint6[12835] = {X 183.6792, Y 19.2349, Z -8.0000, A 0.000, B 0.000, C 0.000 }
gfCNCPoint6[12836] = {X 182.3555, Y 19.6146, Z -8.0000, A 0.000, B 0.000, C 0.000 }
gfCNCPoint6[12837] = {X 181.1074, Y 20.1965, Z -8.0000, A 0.000, B 0.000, C 0.000 }
gfCNCPoint6[12838] = {X 181.0812, Y 20.3299, Z -8.0000, A 0.000, B 0.000, C 0.000 }
gfCNCPoint6[12839] = {X 180.8699, Y 21.2784, Z -8.0000, A 0.000, B 0.000, C 0.000 }
gfCNCPoint6[12840] = {X 180.4402, Y 22.1500, Z -8.0000, A 0.000, B 0.000, C 0.000 }
gfCNCPoint6[12841] = {X 179.8167, Y 22.8952, Z -8.0000, A 0.000, B 0.000, C 0.000 }
gfCNCPoint6[12842] = {X 180.1963, Y 22.9058, Z -8.0000, A 0.000, B 0.000, C 0.000 }
gfCNCPoint6[12843] = {X 182.2705, Y 22.6859, Z -8.0000, A 0.000, B 0.000, C 0.000 }
gfCNCPoint6[12844] = {X 184.3520, Y 22.5520, Z -8.0000, A 0.000, B 0.000, C 0.000 }
gfCNCPoint6[12845] = {X 184.7889, Y 22.5359, Z -8.0000, A 0.000, B 0.000, C 0.000 }
gfCNCPoint6[12846] = {X 185.2258, Y 22.5183, Z -8.0000, A 0.000, B 0.000, C 0.000 }
gfCNCPoint6[12847] = {X 189.1922, Y 22.0013, Z -8.0000, A 0.000, B 0.000, C 0.000 }
gfCNCPoint6[12848] = {X 185.1541, Y 22.6013, Z -8.0000, A 0.000, B 0.000, C 0.000 }
gfCNCPoint6[12849] = {X 185.2292, Y 22.5982, Z -8.0000, A 0.000, B 0.000, C 0.000 }
gfCNCPoint6[12850] = {X 187.5636, Y 22.4756, Z -8.0000, A 0.000, B 0.000, C 0.000 }
gfCNCPoint6[12851] = {X 189.8950, Y 22.3058, Z -8.0000, A 0.000, B 0.000, C 0.000 }
gfCNCPoint6[12852] = {X 190.6493, Y 22.2018, Z -8.0000, A 0.000, B 0.000, C 0.000 }
gfCNCPoint6[12853] = {X 191.3807, Y 21.9897, Z -8.0000, A 0.000, B 0.000, C 0.000 }
gfCNCPoint6[12854] = {X 191.4886, Y 21.4336, Z -8.0000, A 0.000, B 0.000, C 0.000 }
gfCNCPoint6[12855] = {X 191.4045, Y 20.8734, Z -8.0000, A 0.000, B 0.000, C 0.000 }
gfCNCPoint6[12856] = {X 191.1381, Y 20.3734, Z -8.0000, A 0.000, B 0.000, C 0.000 }
gfCNCPoint6[12857] = {X 190.7199, Y 19.9912, Z -8.0000, A 0.000, B 0.000, C 0.000 }
gfCNCPoint6[12858] = {X 189.8090, Y 19.5011, Z -8.0000, A 0.000, B 0.000, C 0.000 }
gfCNCPoint6[12859] = {X 188.8340, Y 19.1560, Z -8.0000, A 0.000, B 0.000, C 0.000 }
gfCNCPoint6[12860] = {X 187.8176, Y 18.9639, Z -8.0000, A 0.000, B 0.000, C 0.000 }
gfCNCPoint6[12861] = {X 186.4284, Y 18.8781, Z -8.0000, A 0.000, B 0.000, C 0.000 }
gfCNCPoint6[12862] = {X 185.0380, Y 18.9426, Z -8.0000, A 0.000, B 0.000, C 0.000 }
gfCNCPoint6[12863] = {X 183.6627, Y 19.1566, Z -8.0000, A 0.000, B 0.000, C 0.000 }
gfCNCPoint6[12864] = {X 182.3100, Y 19.5463, Z -8.0000, A 0.000, B 0.000, C 0.000 }
gfCNCPoint6[12865] = {X 181.0359, Y 20.1451, Z -8.0000, A 0.000, B 0.000, C 0.000 }
gfCNCPoint6[12866] = {X 181.0020, Y 20.3183, Z -8.0000, A 0.000, B 0.000, C 0.000 }
gfCNCPoint6[12867] = {X 180.8538, Y 21.0695, Z -8.0000, A 0.000, B 0.000, C 0.000 }
gfCNCPoint6[12868] = {X 180.5651, Y 21.7787, Z -8.0000, A 0.000, B 0.000, C 0.000 }
gfCNCPoint6[12869] = {X 180.1466, Y 22.4199, Z -8.0000, A 0.000, B 0.000, C 0.000 }
gfCNCPoint6[12870] = {X 179.6136, Y 22.9696, Z -8.0000, A 0.000, B 0.000, C 0.000 }
gfCNCPoint6[12871] = {X 180.2003, Y 22.9859, Z -8.0000, A 0.000, B 0.000, C 0.000 }
gfCNCPoint6[12872] = {X 182.2741, Y 22.7659, Z -8.0000, A 0.000, B 0.000, C 0.000 }
gfCNCPoint6[12873] = {X 184.3552, Y 22.6319, Z -8.0000, A 0.000, B 0.000, C 0.000 }
gfCNCPoint6[12874] = {X 184.7922, Y 22.6159, Z -8.0000, A 0.000, B 0.000, C 0.000 }
gfCNCPoint6[12875] = {X 185.2292, Y 22.5982, Z -8.0000, A 0.000, B 0.000, C 0.000 }
gfCNCPoint6[12876] = {X 185.1445, Y 20.6000, Z -8.0000, A 0.000, B 0.000, C 0.000 }
gfCNCPoint6[12877] = {X 185.1445, Y 20.6000, Z -5.0000, A 0.000, B 0.000, C 0.000 }
gfCNCPoint6[12878] = {X 185.1445, Y 20.6000, Z 11.0000, A 0.000, B 0.000, C 0.000 }
gfCNCPoint6[12879] = {X 186.2252, Y 37.9113, Z 11.0000, A 0.000, B 0.000, C 0.000 }
gfCNCPoint6[12880] = {X 186.2252, Y 37.9113, Z -4.1667, A 0.000, B 0.000, C 0.000 }
gfCNCPoint6[12881] = {X 187.6033, Y 37.8291, Z -4.5366, A 0.000, B 0.000, C 0.000 }
gfCNCPoint6[12882] = {X 189.4365, Y 37.3779, Z -5.0424, A 0.000, B 0.000, C 0.000 }
gfCNCPoint6[12883] = {X 190.1609, Y 37.0645, Z -5.2539, A 0.000, B 0.000, C 0.000 }
gfCNCPoint6[12884] = {X 191.0027, Y 36.7004, Z -5.4997, A 0.000, B 0.000, C 0.000 }
gfCNCPoint6[12885] = {X 191.6870, Y 36.3252, Z -5.7088, A 0.000, B 0.000, C 0.000 }
gfCNCPoint6[12886] = {X 192.4467, Y 35.8114, Z -5.9545, A 0.000, B 0.000, C 0.000 }
gfCNCPoint6[12887] = {X 192.4700, Y 35.2973, Z -6.0924, A 0.000, B 0.000, C 0.000 }
gfCNCPoint6[12888] = {X 192.6308, Y 34.6362, Z -6.2747, A 0.000, B 0.000, C 0.000 }
gfCNCPoint6[12889] = {X 192.8463, Y 34.1688, Z -6.4126, A 0.000, B 0.000, C 0.000 }
gfCNCPoint6[12890] = {X 192.7388, Y 34.1939, Z -6.4422, A 0.000, B 0.000, C 0.000 }
gfCNCPoint6[12891] = {X 191.4058, Y 34.4443, Z -6.8056, A 0.000, B 0.000, C 0.000 }
gfCNCPoint6[12892] = {X 190.5837, Y 34.5501, Z -7.0278, A 0.000, B 0.000, C 0.000 }
gfCNCPoint6[12893] = {X 189.2271, Y 34.6455, Z -7.3921, A 0.000, B 0.000, C 0.000 }
gfCNCPoint6[12894] = {X 186.9628, Y 34.7846, Z -8.0000, A 0.000, B 0.000, C 0.000 }
gfCNCPoint6[12895] = {X 182.5917, Y 35.0530, Z -8.0000, A 0.000, B 0.000, C 0.000 }
gfCNCPoint6[12896] = {X 181.8260, Y 35.1409, Z -8.0000, A 0.000, B 0.000, C 0.000 }
gfCNCPoint6[12897] = {X 181.0738, Y 35.3093, Z -8.0000, A 0.000, B 0.000, C 0.000 }
gfCNCPoint6[12898] = {X 181.0659, Y 35.3830, Z -8.0000, A 0.000, B 0.000, C 0.000 }
gfCNCPoint6[12899] = {X 181.0661, Y 35.4571, Z -8.0000, A 0.000, B 0.000, C 0.000 }
gfCNCPoint6[12900] = {X 181.1585, Y 35.9996, Z -8.0000, A 0.000, B 0.000, C 0.000 }
gfCNCPoint6[12901] = {X 181.4153, Y 36.4863, Z -8.0000, A 0.000, B 0.000, C 0.000 }
gfCNCPoint6[12902] = {X 181.8108, Y 36.8688, Z -8.0000, A 0.000, B 0.000, C 0.000 }
gfCNCPoint6[12903] = {X 182.4283, Y 37.2218, Z -8.0000, A 0.000, B 0.000, C 0.000 }
gfCNCPoint6[12904] = {X 183.0885, Y 37.4862, Z -8.0000, A 0.000, B 0.000, C 0.000 }
gfCNCPoint6[12905] = {X 184.4988, Y 37.8007, Z -8.0000, A 0.000, B 0.000, C 0.000 }
gfCNCPoint6[12906] = {X 185.9392, Y 37.9161, Z -8.0000, A 0.000, B 0.000, C 0.000 }
gfCNCPoint6[12907] = {X 187.3815, Y 37.8301, Z -8.0000, A 0.000, B 0.000, C 0.000 }
gfCNCPoint6[12908] = {X 188.7980, Y 37.5444, Z -8.0000, A 0.000, B 0.000, C 0.000 }
gfCNCPoint6[12909] = {X 190.1609, Y 37.0645, Z -8.0000, A 0.000, B 0.000, C 0.000 }
gfCNCPoint6[12910] = {X 191.3330, Y 36.4913, Z -8.0000, A 0.000, B 0.000, C 0.000 }
gfCNCPoint6[12911] = {X 192.4467, Y 35.8114, Z -8.0000, A 0.000, B 0.000, C 0.000 }
gfCNCPoint6[12912] = {X 192.5669, Y 34.9708, Z -8.0000, A 0.000, B 0.000, C 0.000 }
gfCNCPoint6[12913] = {X 192.8463, Y 34.1688, Z -8.0000, A 0.000, B 0.000, C 0.000 }
gfCNCPoint6[12914] = {X 192.7388, Y 34.1939, Z -8.0000, A 0.000, B 0.000, C 0.000 }
gfCNCPoint6[12915] = {X 190.9895, Y 34.4705, Z -8.0000, A 0.000, B 0.000, C 0.000 }
gfCNCPoint6[12916] = {X 189.2271, Y 34.6455, Z -8.0000, A 0.000, B 0.000, C 0.000 }
gfCNCPoint6[12917] = {X 186.9628, Y 34.7846, Z -8.0000, A 0.000, B 0.000, C 0.000 }
gfCNCPoint6[12918] = {X 190.9566, Y 34.8085, Z -8.0000, A 0.000, B 0.000, C 0.000 }
gfCNCPoint6[12919] = {X 186.9579, Y 34.7047, Z -8.0000, A 0.000, B 0.000, C 0.000 }
gfCNCPoint6[12920] = {X 182.5868, Y 34.9731, Z -8.0000, A 0.000, B 0.000, C 0.000 }
gfCNCPoint6[12921] = {X 181.7884, Y 35.0661, Z -8.0000, A 0.000, B 0.000, C 0.000 }
gfCNCPoint6[12922] = {X 181.0048, Y 35.2457, Z -8.0000, A 0.000, B 0.000, C 0.000 }
gfCNCPoint6[12923] = {X 180.9883, Y 35.3487, Z -8.0000, A 0.000, B 0.000, C 0.000 }
gfCNCPoint6[12924] = {X 180.9861, Y 35.4529, Z -8.0000, A 0.000, B 0.000, C 0.000 }
gfCNCPoint6[12925] = {X 181.0818, Y 36.0224, Z -8.0000, A 0.000, B 0.000, C 0.000 }
gfCNCPoint6[12926] = {X 181.3506, Y 36.5334, Z -8.0000, A 0.000, B 0.000, C 0.000 }
gfCNCPoint6[12927] = {X 181.7657, Y 36.9349, Z -8.0000, A 0.000, B 0.000, C 0.000 }
gfCNCPoint6[12928] = {X 182.3935, Y 37.2938, Z -8.0000, A 0.000, B 0.000, C 0.000 }
gfCNCPoint6[12929] = {X 183.0649, Y 37.5626, Z -8.0000, A 0.000, B 0.000, C 0.000 }
gfCNCPoint6[12930] = {X 184.4862, Y 37.8797, Z -8.0000, A 0.000, B 0.000, C 0.000 }
gfCNCPoint6[12931] = {X 185.9378, Y 37.9960, Z -8.0000, A 0.000, B 0.000, C 0.000 }
gfCNCPoint6[12932] = {X 187.3915, Y 37.9094, Z -8.0000, A 0.000, B 0.000, C 0.000 }
gfCNCPoint6[12933] = {X 188.8190, Y 37.6215, Z -8.0000, A 0.000, B 0.000, C 0.000 }
gfCNCPoint6[12934] = {X 190.1927, Y 37.1379, Z -8.0000, A 0.000, B 0.000, C 0.000 }
gfCNCPoint6[12935] = {X 191.3892, Y 36.5517, Z -8.0000, A 0.000, B 0.000, C 0.000 }
gfCNCPoint6[12936] = {X 192.5250, Y 35.8550, Z -8.0000, A 0.000, B 0.000, C 0.000 }
gfCNCPoint6[12937] = {X 192.6601, Y 34.9281, Z -8.0000, A 0.000, B 0.000, C 0.000 }
gfCNCPoint6[12938] = {X 192.9918, Y 34.0521, Z -8.0000, A 0.000, B 0.000, C 0.000 }
gfCNCPoint6[12939] = {X 192.7315, Y 34.1138, Z -8.0000, A 0.000, B 0.000, C 0.000 }
gfCNCPoint6[12940] = {X 190.9841, Y 34.3905, Z -8.0000, A 0.000, B 0.000, C 0.000 }
gfCNCPoint6[12941] = {X 189.2236, Y 34.5656, Z -8.0000, A 0.000, B 0.000, C 0.000 }
gfCNCPoint6[12942] = {X 186.9579, Y 34.7047, Z -8.0000, A 0.000, B 0.000, C 0.000 }
gfCNCPoint6[12943] = {X 183.0020, Y 35.2969, Z -8.0000, A 0.000, B 0.000, C 0.000 }
gfCNCPoint6[12944] = {X 190.9517, Y 34.7286, Z -8.0000, A 0.000, B 0.000, C 0.000 }
gfCNCPoint6[12945] = {X 186.9530, Y 34.6249, Z -8.0000, A 0.000, B 0.000, C 0.000 }
gfCNCPoint6[12946] = {X 182.5819, Y 34.8933, Z -8.0000, A 0.000, B 0.000, C 0.000 }
gfCNCPoint6[12947] = {X 181.7524, Y 34.9912, Z -8.0000, A 0.000, B 0.000, C 0.000 }
gfCNCPoint6[12948] = {X 180.9390, Y 35.1815, Z -8.0000, A 0.000, B 0.000, C 0.000 }
gfCNCPoint6[12949] = {X 180.9112, Y 35.3169, Z -8.0000, A 0.000, B 0.000, C 0.000 }
gfCNCPoint6[12950] = {X 180.9061, Y 35.4551, Z -8.0000, A 0.000, B 0.000, C 0.000 }
gfCNCPoint6[12951] = {X 181.0064, Y 36.0492, Z -8.0000, A 0.000, B 0.000, C 0.000 }
gfCNCPoint6[12952] = {X 181.2873, Y 36.5823, Z -8.0000, A 0.000, B 0.000, C 0.000 }
gfCNCPoint6[12953] = {X 181.7206, Y 37.0009, Z -8.0000, A 0.000, B 0.000, C 0.000 }
gfCNCPoint6[12954] = {X 182.3587, Y 37.3659, Z -8.0000, A 0.000, B 0.000, C 0.000 }
gfCNCPoint6[12955] = {X 183.0412, Y 37.6390, Z -8.0000, A 0.000, B 0.000, C 0.000 }
gfCNCPoint6[12956] = {X 184.4736, Y 37.9587, Z -8.0000, A 0.000, B 0.000, C 0.000 }
gfCNCPoint6[12957] = {X 185.9365, Y 38.0760, Z -8.0000, A 0.000, B 0.000, C 0.000 }
gfCNCPoint6[12958] = {X 187.4015, Y 37.9888, Z -8.0000, A 0.000, B 0.000, C 0.000 }
gfCNCPoint6[12959] = {X 188.8401, Y 37.6987, Z -8.0000, A 0.000, B 0.000, C 0.000 }
gfCNCPoint6[12960] = {X 190.2244, Y 37.2114, Z -8.0000, A 0.000, B 0.000, C 0.000 }
gfCNCPoint6[12961] = {X 191.4456, Y 36.6119, Z -8.0000, A 0.000, B 0.000, C 0.000 }
gfCNCPoint6[12962] = {X 192.6036, Y 35.8981, Z -8.0000, A 0.000, B 0.000, C 0.000 }
gfCNCPoint6[12963] = {X 192.6772, Y 35.2167, Z -8.0000, A 0.000, B 0.000, C 0.000 }
gfCNCPoint6[12964] = {X 192.8596, Y 34.5560, Z -8.0000, A 0.000, B 0.000, C 0.000 }
gfCNCPoint6[12965] = {X 193.1461, Y 33.9333, Z -8.0000, A 0.000, B 0.000, C 0.000 }
gfCNCPoint6[12966] = {X 192.7149, Y 34.0356, Z -8.0000, A 0.000, B 0.000, C 0.000 }
gfCNCPoint6[12967] = {X 190.9731, Y 34.3113, Z -8.0000, A 0.000, B 0.000, C 0.000 }
gfCNCPoint6[12968] = {X 189.2183, Y 34.4858, Z -8.0000, A 0.000, B 0.000, C 0.000 }
gfCNCPoint6[12969] = {X 186.9530, Y 34.6249, Z -8.0000, A 0.000, B 0.000, C 0.000 }
gfCNCPoint6[12970] = {X 182.9971, Y 35.2170, Z -8.0000, A 0.000, B 0.000, C 0.000 }
gfCNCPoint6[12971] = {X 190.9468, Y 34.6488, Z -8.0000, A 0.000, B 0.000, C 0.000 }
gfCNCPoint6[12972] = {X 186.9481, Y 34.5450, Z -8.0000, A 0.000, B 0.000, C 0.000 }
gfCNCPoint6[12973] = {X 182.5770, Y 34.8134, Z -8.0000, A 0.000, B 0.000, C 0.000 }
gfCNCPoint6[12974] = {X 181.7176, Y 34.9161, Z -8.0000, A 0.000, B 0.000, C 0.000 }
gfCNCPoint6[12975] = {X 180.8757, Y 35.1169, Z -8.0000, A 0.000, B 0.000, C 0.000 }
gfCNCPoint6[12976] = {X 180.8348, Y 35.2847, Z -8.0000, A 0.000, B 0.000, C 0.000 }
gfCNCPoint6[12977] = {X 180.8261, Y 35.4572, Z -8.0000, A 0.000, B 0.000, C 0.000 }
gfCNCPoint6[12978] = {X 180.9310, Y 36.0760, Z -8.0000, A 0.000, B 0.000, C 0.000 }
gfCNCPoint6[12979] = {X 181.2239, Y 36.6311, Z -8.0000, A 0.000, B 0.000, C 0.000 }
gfCNCPoint6[12980] = {X 181.6754, Y 37.0670, Z -8.0000, A 0.000, B 0.000, C 0.000 }
gfCNCPoint6[12981] = {X 182.3239, Y 37.4379, Z -8.0000, A 0.000, B 0.000, C 0.000 }
gfCNCPoint6[12982] = {X 183.0175, Y 37.7155, Z -8.0000, A 0.000, B 0.000, C 0.000 }
gfCNCPoint6[12983] = {X 184.4609, Y 38.0377, Z -8.0000, A 0.000, B 0.000, C 0.000 }
gfCNCPoint6[12984] = {X 185.9351, Y 38.1560, Z -8.0000, A 0.000, B 0.000, C 0.000 }
gfCNCPoint6[12985] = {X 187.4114, Y 38.0682, Z -8.0000, A 0.000, B 0.000, C 0.000 }
gfCNCPoint6[12986] = {X 188.8612, Y 37.7759, Z -8.0000, A 0.000, B 0.000, C 0.000 }
gfCNCPoint6[12987] = {X 190.2562, Y 37.2848, Z -8.0000, A 0.000, B 0.000, C 0.000 }
gfCNCPoint6[12988] = {X 191.5022, Y 36.6720, Z -8.0000, A 0.000, B 0.000, C 0.000 }
gfCNCPoint6[12989] = {X 192.6827, Y 35.9409, Z -8.0000, A 0.000, B 0.000, C 0.000 }
gfCNCPoint6[12990] = {X 192.7625, Y 35.1972, Z -8.0000, A 0.000, B 0.000, C 0.000 }
gfCNCPoint6[12991] = {X 192.9741, Y 34.4799, Z -8.0000, A 0.000, B 0.000, C 0.000 }
gfCNCPoint6[12992] = {X 193.3108, Y 33.8121, Z -8.0000, A 0.000, B 0.000, C 0.000 }
gfCNCPoint6[12993] = {X 192.6982, Y 33.9573, Z -8.0000, A 0.000, B 0.000, C 0.000 }
gfCNCPoint6[12994] = {X 190.9621, Y 34.2320, Z -8.0000, A 0.000, B 0.000, C 0.000 }
gfCNCPoint6[12995] = {X 189.2131, Y 34.4059, Z -8.0000, A 0.000, B 0.000, C 0.000 }
gfCNCPoint6[12996] = {X 186.9481, Y 34.5450, Z -8.0000, A 0.000, B 0.000, C 0.000 }
gfCNCPoint6[12997] = {X 182.9922, Y 35.1372, Z -8.0000, A 0.000, B 0.000, C 0.000 }
gfCNCPoint6[12998] = {X 190.9419, Y 34.5689, Z -8.0000, A 0.000, B 0.000, C 0.000 }
gfCNCPoint6[12999] = {X 186.9432, Y 34.4652, Z -8.0000, A 0.000, B 0.000, C 0.000 }
gfCNCPoint6[13000] = {X 182.5721, Y 34.7336, Z -8.0000, A 0.000, B 0.000, C 0.000 }
gfCNCPoint6[13001] = {X 181.6839, Y 34.8409, Z -8.0000, A 0.000, B 0.000, C 0.000 }
gfCNCPoint6[13002] = {X 180.8144, Y 35.0518, Z -8.0000, A 0.000, B 0.000, C 0.000 }
gfCNCPoint6[13003] = {X 180.7590, Y 35.2520, Z -8.0000, A 0.000, B 0.000, C 0.000 }
gfCNCPoint6[13004] = {X 180.7461, Y 35.4593, Z -8.0000, A 0.000, B 0.000, C 0.000 }
gfCNCPoint6[13005] = {X 180.8556, Y 36.1028, Z -8.0000, A 0.000, B 0.000, C 0.000 }
gfCNCPoint6[13006] = {X 181.1605, Y 36.6799, Z -8.0000, A 0.000, B 0.000, C 0.000 }
gfCNCPoint6[13007] = {X 181.6303, Y 37.1331, Z -8.0000, A 0.000, B 0.000, C 0.000 }
gfCNCPoint6[13008] = {X 182.2892, Y 37.5100, Z -8.0000, A 0.000, B 0.000, C 0.000 }
gfCNCPoint6[13009] = {X 182.9939, Y 37.7919, Z -8.0000, A 0.000, B 0.000, C 0.000 }
gfCNCPoint6[13010] = {X 184.4483, Y 38.1167, Z -8.0000, A 0.000, B 0.000, C 0.000 }
gfCNCPoint6[13011] = {X 185.9338, Y 38.2360, Z -8.0000, A 0.000, B 0.000, C 0.000 }
gfCNCPoint6[13012] = {X 187.4214, Y 38.1476, Z -8.0000, A 0.000, B 0.000, C 0.000 }
gfCNCPoint6[13013] = {X 188.8823, Y 37.8531, Z -8.0000, A 0.000, B 0.000, C 0.000 }
gfCNCPoint6[13014] = {X 190.2879, Y 37.3582, Z -8.0000, A 0.000, B 0.000, C 0.000 }
gfCNCPoint6[13015] = {X 191.5591, Y 36.7320, Z -8.0000, A 0.000, B 0.000, C 0.000 }
gfCNCPoint6[13016] = {X 192.7622, Y 35.9832, Z -8.0000, A 0.000, B 0.000, C 0.000 }
gfCNCPoint6[13017] = {X 192.8357, Y 35.2397, Z -8.0000, A 0.000, B 0.000, C 0.000 }
gfCNCPoint6[13018] = {X 193.0435, Y 34.5221, Z -8.0000, A 0.000, B 0.000, C 0.000 }
gfCNCPoint6[13019] = {X 193.3787, Y 33.8544, Z -8.0000, A 0.000, B 0.000, C 0.000 }
gfCNCPoint6[13020] = {X 193.4220, Y 33.7864, Z -8.0000, A 0.000, B 0.000, C 0.000 }
gfCNCPoint6[13021] = {X 193.4665, Y 33.7193, Z -8.0000, A 0.000, B 0.000, C 0.000 }
gfCNCPoint6[13022] = {X 193.3658, Y 33.7168, Z -8.0000, A 0.000, B 0.000, C 0.000 }
gfCNCPoint6[13023] = {X 192.6816, Y 33.8790, Z -8.0000, A 0.000, B 0.000, C 0.000 }
gfCNCPoint6[13024] = {X 190.9512, Y 34.1528, Z -8.0000, A 0.000, B 0.000, C 0.000 }
gfCNCPoint6[13025] = {X 189.2078, Y 34.3261, Z -8.0000, A 0.000, B 0.000, C 0.000 }
gfCNCPoint6[13026] = {X 186.9432, Y 34.4652, Z -8.0000, A 0.000, B 0.000, C 0.000 }
gfCNCPoint6[13027] = {X 182.9873, Y 35.0573, Z -8.0000, A 0.000, B 0.000, C 0.000 }
gfCNCPoint6[13028] = {X 190.9369, Y 34.4891, Z -8.0000, A 0.000, B 0.000, C 0.000 }
gfCNCPoint6[13029] = {X 186.9383, Y 34.3853, Z -8.0000, A 0.000, B 0.000, C 0.000 }
gfCNCPoint6[13030] = {X 182.5672, Y 34.6537, Z -8.0000, A 0.000, B 0.000, C 0.000 }
gfCNCPoint6[13031] = {X 181.6510, Y 34.7655, Z -8.0000, A 0.000, B 0.000, C 0.000 }
gfCNCPoint6[13032] = {X 180.7549, Y 34.9865, Z -8.0000, A 0.000, B 0.000, C 0.000 }
gfCNCPoint6[13033] = {X 180.6836, Y 35.2189, Z -8.0000, A 0.000, B 0.000, C 0.000 }
gfCNCPoint6[13034] = {X 180.6661, Y 35.4613, Z -8.0000, A 0.000, B 0.000, C 0.000 }
gfCNCPoint6[13035] = {X 180.7802, Y 36.1295, Z -8.0000, A 0.000, B 0.000, C 0.000 }
gfCNCPoint6[13036] = {X 181.0971, Y 36.7288, Z -8.0000, A 0.000, B 0.000, C 0.000 }
gfCNCPoint6[13037] = {X 181.5852, Y 37.1992, Z -8.0000, A 0.000, B 0.000, C 0.000 }
gfCNCPoint6[13038] = {X 182.2544, Y 37.5820, Z -8.0000, A 0.000, B 0.000, C 0.000 }
gfCNCPoint6[13039] = {X 182.9702, Y 37.8683, Z -8.0000, A 0.000, B 0.000, C 0.000 }
gfCNCPoint6[13040] = {X 184.4357, Y 38.1957, Z -8.0000, A 0.000, B 0.000, C 0.000 }
gfCNCPoint6[13041] = {X 185.9324, Y 38.3160, Z -8.0000, A 0.000, B 0.000, C 0.000 }
gfCNCPoint6[13042] = {X 187.4314, Y 38.2269, Z -8.0000, A 0.000, B 0.000, C 0.000 }
gfCNCPoint6[13043] = {X 188.9033, Y 37.9302, Z -8.0000, A 0.000, B 0.000, C 0.000 }
gfCNCPoint6[13044] = {X 190.3197, Y 37.4316, Z -8.0000, A 0.000, B 0.000, C 0.000 }
gfCNCPoint6[13045] = {X 191.6163, Y 36.7917, Z -8.0000, A 0.000, B 0.000, C 0.000 }
gfCNCPoint6[13046] = {X 192.8422, Y 36.0250, Z -8.0000, A 0.000, B 0.000, C 0.000 }
gfCNCPoint6[13047] = {X 192.9290, Y 35.1818, Z -8.0000, A 0.000, B 0.000, C 0.000 }
gfCNCPoint6[13048] = {X 193.1917, Y 34.3757, Z -8.0000, A 0.000, B 0.000, C 0.000 }
gfCNCPoint6[13049] = {X 193.6183, Y 33.6431, Z -8.0000, A 0.000, B 0.000, C 0.000 }
gfCNCPoint6[13050] = {X 193.3575, Y 33.6366, Z -8.0000, A 0.000, B 0.000, C 0.000 }
gfCNCPoint6[13051] = {X 192.6650, Y 33.8007, Z -8.0000, A 0.000, B 0.000, C 0.000 }
gfCNCPoint6[13052] = {X 190.9402, Y 34.0735, Z -8.0000, A 0.000, B 0.000, C 0.000 }
gfCNCPoint6[13053] = {X 189.2026, Y 34.2463, Z -8.0000, A 0.000, B 0.000, C 0.000 }
gfCNCPoint6[13054] = {X 186.9383, Y 34.3853, Z -8.0000, A 0.000, B 0.000, C 0.000 }
gfCNCPoint6[13055] = {X 182.9458, Y 34.6305, Z -8.0000, A 0.000, B 0.000, C 0.000 }
gfCNCPoint6[13056] = {X 182.9458, Y 34.6305, Z -5.0000, A 0.000, B 0.000, C 0.000 }
gfCNCPoint6[13057] = {X 182.9458, Y 34.6305, Z 11.0000, A 0.000, B 0.000, C 0.000 }
gfCNCPoint6[13058] = {X 165.6772, Y 73.8165, Z 11.0000, A 0.000, B 0.000, C 0.000 }
gfCNCPoint6[13059] = {X 165.6772, Y 73.8165, Z -4.1667, A 0.000, B 0.000, C 0.000 }
gfCNCPoint6[13060] = {X 161.3996, Y 78.5670, Z -5.8796, A 0.000, B 0.000, C 0.000 }
gfCNCPoint6[13061] = {X 169.3132, Y 78.5670, Z -8.0000, A 0.000, B 0.000, C 0.000 }
gfCNCPoint6[13062] = {X 169.3132, Y 76.1670, Z -8.0000, A 0.000, B 0.000, C 0.000 }
gfCNCPoint6[13063] = {X 171.8361, Y 76.1670, Z -8.0000, A 0.000, B 0.000, C 0.000 }
gfCNCPoint6[13064] = {X 169.3147, Y 73.3634, Z -8.0000, A 0.000, B 0.000, C 0.000 }
gfCNCPoint6[13065] = {X 166.7903, Y 76.1670, Z -8.0000, A 0.000, B 0.000, C 0.000 }
gfCNCPoint6[13066] = {X 169.3132, Y 76.1670, Z -8.0000, A 0.000, B 0.000, C 0.000 }
gfCNCPoint6[13067] = {X 169.3132, Y 78.5670, Z -8.0000, A 0.000, B 0.000, C 0.000 }
gfCNCPoint6[13068] = {X 177.2224, Y 78.5670, Z -8.0000, A 0.000, B 0.000, C 0.000 }
gfCNCPoint6[13069] = {X 169.3158, Y 69.7756, Z -8.0000, A 0.000, B 0.000, C 0.000 }
gfCNCPoint6[13070] = {X 161.3996, Y 78.5670, Z -8.0000, A 0.000, B 0.000, C 0.000 }
gfCNCPoint6[13071] = {X 169.3132, Y 78.5670, Z -8.0000, A 0.000, B 0.000, C 0.000 }
gfCNCPoint6[13072] = {X 169.3132, Y 74.6470, Z -8.0000, A 0.000, B 0.000, C 0.000 }
gfCNCPoint6[13073] = {X 169.3132, Y 78.6470, Z -8.0000, A 0.000, B 0.000, C 0.000 }
gfCNCPoint6[13074] = {X 177.4019, Y 78.6470, Z -8.0000, A 0.000, B 0.000, C 0.000 }
gfCNCPoint6[13075] = {X 169.3159, Y 69.6560, Z -8.0000, A 0.000, B 0.000, C 0.000 }
gfCNCPoint6[13076] = {X 161.2199, Y 78.6470, Z -8.0000, A 0.000, B 0.000, C 0.000 }
gfCNCPoint6[13077] = {X 169.3132, Y 78.6470, Z -8.0000, A 0.000, B 0.000, C 0.000 }
gfCNCPoint6[13078] = {X 169.3132, Y 74.6470, Z -8.0000, A 0.000, B 0.000, C 0.000 }
gfCNCPoint6[13079] = {X 169.3132, Y 74.7270, Z -8.0000, A 0.000, B 0.000, C 0.000 }
gfCNCPoint6[13080] = {X 169.3132, Y 78.7270, Z -8.0000, A 0.000, B 0.000, C 0.000 }
gfCNCPoint6[13081] = {X 177.5814, Y 78.7270, Z -8.0000, A 0.000, B 0.000, C 0.000 }
gfCNCPoint6[13082] = {X 169.3159, Y 69.5364, Z -8.0000, A 0.000, B 0.000, C 0.000 }
gfCNCPoint6[13083] = {X 161.0403, Y 78.7270, Z -8.0000, A 0.000, B 0.000, C 0.000 }
gfCNCPoint6[13084] = {X 169.3132, Y 78.7270, Z -8.0000, A 0.000, B 0.000, C 0.000 }
gfCNCPoint6[13085] = {X 169.3132, Y 74.7270, Z -8.0000, A 0.000, B 0.000, C 0.000 }
gfCNCPoint6[13086] = {X 169.3132, Y 74.8070, Z -8.0000, A 0.000, B 0.000, C 0.000 }
gfCNCPoint6[13087] = {X 169.3132, Y 78.8070, Z -8.0000, A 0.000, B 0.000, C 0.000 }
gfCNCPoint6[13088] = {X 177.7610, Y 78.8070, Z -8.0000, A 0.000, B 0.000, C 0.000 }
gfCNCPoint6[13089] = {X 169.3159, Y 69.4168, Z -8.0000, A 0.000, B 0.000, C 0.000 }
gfCNCPoint6[13090] = {X 160.8606, Y 78.8070, Z -8.0000, A 0.000, B 0.000, C 0.000 }
gfCNCPoint6[13091] = {X 169.3132, Y 78.8070, Z -8.0000, A 0.000, B 0.000, C 0.000 }
gfCNCPoint6[13092] = {X 169.3132, Y 74.8070, Z -8.0000, A 0.000, B 0.000, C 0.000 }
gfCNCPoint6[13093] = {X 169.3132, Y 74.8870, Z -8.0000, A 0.000, B 0.000, C 0.000 }
gfCNCPoint6[13094] = {X 169.3132, Y 78.8870, Z -8.0000, A 0.000, B 0.000, C 0.000 }
gfCNCPoint6[13095] = {X 177.9405, Y 78.8870, Z -8.0000, A 0.000, B 0.000, C 0.000 }
gfCNCPoint6[13096] = {X 169.3160, Y 69.2972, Z -8.0000, A 0.000, B 0.000, C 0.000 }
gfCNCPoint6[13097] = {X 160.6809, Y 78.8870, Z -8.0000, A 0.000, B 0.000, C 0.000 }
gfCNCPoint6[13098] = {X 169.3132, Y 78.8870, Z -8.0000, A 0.000, B 0.000, C 0.000 }
gfCNCPoint6[13099] = {X 169.3132, Y 74.8870, Z -8.0000, A 0.000, B 0.000, C 0.000 }
gfCNCPoint6[13100] = {X 169.3132, Y 74.9670, Z -8.0000, A 0.000, B 0.000, C 0.000 }
gfCNCPoint6[13101] = {X 169.3132, Y 78.9670, Z -8.0000, A 0.000, B 0.000, C 0.000 }
gfCNCPoint6[13102] = {X 178.1201, Y 78.9670, Z -8.0000, A 0.000, B 0.000, C 0.000 }
gfCNCPoint6[13103] = {X 169.3160, Y 69.1776, Z -8.0000, A 0.000, B 0.000, C 0.000 }
gfCNCPoint6[13104] = {X 160.5012, Y 78.9670, Z -8.0000, A 0.000, B 0.000, C 0.000 }
gfCNCPoint6[13105] = {X 169.3132, Y 78.9670, Z -8.0000, A 0.000, B 0.000, C 0.000 }
gfCNCPoint6[13106] = {X 169.3132, Y 74.9670, Z -8.0000, A 0.000, B 0.000, C 0.000 }
gfCNCPoint6[13107] = {X 169.3132, Y 74.9670, Z -5.0000, A 0.000, B 0.000, C 0.000 }
gfCNCPoint6[13108] = {X 169.3132, Y 74.9670, Z 11.0000, A 0.000, B 0.000, C 0.000 }
gfCNCPoint6[13109] = {X 11.7076, Y 37.8754, Z 11.0000, A 0.000, B 0.000, C 0.000 }
gfCNCPoint6[13110] = {X 11.7076, Y 37.8754, Z -4.1667, A 0.000, B 0.000, C 0.000 }
gfCNCPoint6[13111] = {X 12.5083, Y 37.9478, Z -4.3821, A 0.000, B 0.000, C 0.000 }
gfCNCPoint6[13112] = {X 14.1614, Y 37.8334, Z -4.8261, A 0.000, B 0.000, C 0.000 }
gfCNCPoint6[13113] = {X 15.7755, Y 37.4584, Z -5.2701, A 0.000, B 0.000, C 0.000 }
gfCNCPoint6[13114] = {X 16.5080, Y 37.1626, Z -5.4818, A 0.000, B 0.000, C 0.000 }
gfCNCPoint6[13115] = {X 17.3401, Y 36.8265, Z -5.7222, A 0.000, B 0.000, C 0.000 }
gfCNCPoint6[13116] = {X 18.2927, Y 36.3173, Z -6.0117, A 0.000, B 0.000, C 0.000 }
gfCNCPoint6[13117] = {X 19.0345, Y 35.8121, Z -6.2521, A 0.000, B 0.000, C 0.000 }
gfCNCPoint6[13118] = {X 19.0577, Y 35.2980, Z -6.3900, A 0.000, B 0.000, C 0.000 }
gfCNCPoint6[13119] = {X 19.2187, Y 34.6363, Z -6.5725, A 0.000, B 0.000, C 0.000 }
gfCNCPoint6[13120] = {X 19.4341, Y 34.1689, Z -6.7104, A 0.000, B 0.000, C 0.000 }
gfCNCPoint6[13121] = {X 18.2048, Y 34.4171, Z -7.0465, A 0.000, B 0.000, C 0.000 }
gfCNCPoint6[13122] = {X 17.3615, Y 34.5318, Z -7.2745, A 0.000, B 0.000, C 0.000 }
gfCNCPoint6[13123] = {X 16.1106, Y 34.6209, Z -7.6105, A 0.000, B 0.000, C 0.000 }
gfCNCPoint6[13124] = {X 15.3858, Y 34.6747, Z -7.8053, A 0.000, B 0.000, C 0.000 }
gfCNCPoint6[13125] = {X 14.6607, Y 34.7242, Z -8.0000, A 0.000, B 0.000, C 0.000 }
gfCNCPoint6[13126] = {X 12.2606, Y 34.8768, Z -8.0000, A 0.000, B 0.000, C 0.000 }
gfCNCPoint6[13127] = {X 9.8591, Y 35.0065, Z -8.0000, A 0.000, B 0.000, C 0.000 }
gfCNCPoint6[13128] = {X 8.7542, Y 35.0964, Z -8.0000, A 0.000, B 0.000, C 0.000 }
gfCNCPoint6[13129] = {X 7.6664, Y 35.3101, Z -8.0000, A 0.000, B 0.000, C 0.000 }
gfCNCPoint6[13130] = {X 7.6569, Y 35.3716, Z -8.0000, A 0.000, B 0.000, C 0.000 }
gfCNCPoint6[13131] = {X 7.6536, Y 35.4337, Z -8.0000, A 0.000, B 0.000, C 0.000 }
gfCNCPoint6[13132] = {X 7.7540, Y 36.0255, Z -8.0000, A 0.000, B 0.000, C 0.000 }
gfCNCPoint6[13133] = {X 8.0478, Y 36.5489, Z -8.0000, A 0.000, B 0.000, C 0.000 }
gfCNCPoint6[13134] = {X 8.5006, Y 36.9430, Z -8.0000, A 0.000, B 0.000, C 0.000 }
gfCNCPoint6[13135] = {X 9.2713, Y 37.3343, Z -8.0000, A 0.000, B 0.000, C 0.000 }
gfCNCPoint6[13136] = {X 10.0917, Y 37.6065, Z -8.0000, A 0.000, B 0.000, C 0.000 }
gfCNCPoint6[13137] = {X 11.3769, Y 37.8440, Z -8.0000, A 0.000, B 0.000, C 0.000 }
gfCNCPoint6[13138] = {X 12.6818, Y 37.9182, Z -8.0000, A 0.000, B 0.000, C 0.000 }
gfCNCPoint6[13139] = {X 13.9856, Y 37.8280, Z -8.0000, A 0.000, B 0.000, C 0.000 }
gfCNCPoint6[13140] = {X 15.2678, Y 37.5748, Z -8.0000, A 0.000, B 0.000, C 0.000 }
gfCNCPoint6[13141] = {X 16.5080, Y 37.1626, Z -8.0000, A 0.000, B 0.000, C 0.000 }
gfCNCPoint6[13142] = {X 17.8074, Y 36.5550, Z -8.0000, A 0.000, B 0.000, C 0.000 }
gfCNCPoint6[13143] = {X 19.0345, Y 35.8121, Z -8.0000, A 0.000, B 0.000, C 0.000 }
gfCNCPoint6[13144] = {X 19.1546, Y 34.9712, Z -8.0000, A 0.000, B 0.000, C 0.000 }
gfCNCPoint6[13145] = {X 19.4341, Y 34.1689, Z -8.0000, A 0.000, B 0.000, C 0.000 }
gfCNCPoint6[13146] = {X 17.7796, Y 34.4482, Z -8.0000, A 0.000, B 0.000, C 0.000 }
gfCNCPoint6[13147] = {X 16.1106, Y 34.6209, Z -8.0000, A 0.000, B 0.000, C 0.000 }
gfCNCPoint6[13148] = {X 15.3857, Y 34.6736, Z -8.0000, A 0.000, B 0.000, C 0.000 }
gfCNCPoint6[13149] = {X 14.6607, Y 34.7242, Z -8.0000, A 0.000, B 0.000, C 0.000 }
gfCNCPoint6[13150] = {X 18.6546, Y 34.7204, Z -8.0000, A 0.000, B 0.000, C 0.000 }
gfCNCPoint6[13151] = {X 14.6553, Y 34.6444, Z -8.0000, A 0.000, B 0.000, C 0.000 }
gfCNCPoint6[13152] = {X 12.2588, Y 34.7968, Z -8.0000, A 0.000, B 0.000, C 0.000 }
gfCNCPoint6[13153] = {X 9.8610, Y 34.9265, Z -8.0000, A 0.000, B 0.000, C 0.000 }
gfCNCPoint6[13154] = {X 8.7214, Y 35.0202, Z -8.0000, A 0.000, B 0.000, C 0.000 }
gfCNCPoint6[13155] = {X 7.6001, Y 35.2446, Z -8.0000, A 0.000, B 0.000, C 0.000 }
gfCNCPoint6[13156] = {X 7.5804, Y 35.3381, Z -8.0000, A 0.000, B 0.000, C 0.000 }
gfCNCPoint6[13157] = {X 7.5736, Y 35.4334, Z -8.0000, A 0.000, B 0.000, C 0.000 }
gfCNCPoint6[13158] = {X 7.6786, Y 36.0522, Z -8.0000, A 0.000, B 0.000, C 0.000 }
gfCNCPoint6[13159] = {X 7.9857, Y 36.5994, Z -8.0000, A 0.000, B 0.000, C 0.000 }
gfCNCPoint6[13160] = {X 8.4591, Y 37.0114, Z -8.0000, A 0.000, B 0.000, C 0.000 }
gfCNCPoint6[13161] = {X 9.2405, Y 37.4081, Z -8.0000, A 0.000, B 0.000, C 0.000 }
gfCNCPoint6[13162] = {X 10.0722, Y 37.6841, Z -8.0000, A 0.000, B 0.000, C 0.000 }
gfCNCPoint6[13163] = {X 11.3673, Y 37.9234, Z -8.0000, A 0.000, B 0.000, C 0.000 }
gfCNCPoint6[13164] = {X 12.6822, Y 37.9982, Z -8.0000, A 0.000, B 0.000, C 0.000 }
gfCNCPoint6[13165] = {X 13.9961, Y 37.9073, Z -8.0000, A 0.000, B 0.000, C 0.000 }
gfCNCPoint6[13166] = {X 15.2882, Y 37.6521, Z -8.0000, A 0.000, B 0.000, C 0.000 }
gfCNCPoint6[13167] = {X 16.5380, Y 37.2367, Z -8.0000, A 0.000, B 0.000, C 0.000 }
gfCNCPoint6[13168] = {X 17.8629, Y 36.6161, Z -8.0000, A 0.000, B 0.000, C 0.000 }
gfCNCPoint6[13169] = {X 19.1128, Y 35.8555, Z -8.0000, A 0.000, B 0.000, C 0.000 }
gfCNCPoint6[13170] = {X 19.2470, Y 34.9316, Z -8.0000, A 0.000, B 0.000, C 0.000 }
gfCNCPoint6[13171] = {X 19.5766, Y 34.0580, Z -8.0000, A 0.000, B 0.000, C 0.000 }
gfCNCPoint6[13172] = {X 17.8488, Y 34.3579, Z -8.0000, A 0.000, B 0.000, C 0.000 }
gfCNCPoint6[13173] = {X 16.1048, Y 34.5411, Z -8.0000, A 0.000, B 0.000, C 0.000 }
gfCNCPoint6[13174] = {X 15.3801, Y 34.5938, Z -8.0000, A 0.000, B 0.000, C 0.000 }
gfCNCPoint6[13175] = {X 14.6553, Y 34.6444, Z -8.0000, A 0.000, B 0.000, C 0.000 }
gfCNCPoint6[13176] = {X 10.7036, Y 35.2641, Z -8.0000, A 0.000, B 0.000, C 0.000 }
gfCNCPoint6[13177] = {X 18.6491, Y 34.6406, Z -8.0000, A 0.000, B 0.000, C 0.000 }
gfCNCPoint6[13178] = {X 14.6498, Y 34.5646, Z -8.0000, A 0.000, B 0.000, C 0.000 }
gfCNCPoint6[13179] = {X 12.2546, Y 34.7170, Z -8.0000, A 0.000, B 0.000, C 0.000 }
gfCNCPoint6[13180] = {X 9.8581, Y 34.8465, Z -8.0000, A 0.000, B 0.000, C 0.000 }
gfCNCPoint6[13181] = {X 8.6878, Y 34.9442, Z -8.0000, A 0.000, B 0.000, C 0.000 }
gfCNCPoint6[13182] = {X 7.5371, Y 35.1785, Z -8.0000, A 0.000, B 0.000, C 0.000 }
gfCNCPoint6[13183] = {X 7.5047, Y 35.3040, Z -8.0000, A 0.000, B 0.000, C 0.000 }
gfCNCPoint6[13184] = {X 7.4936, Y 35.4332, Z -8.0000, A 0.000, B 0.000, C 0.000 }
gfCNCPoint6[13185] = {X 7.6032, Y 36.0788, Z -8.0000, A 0.000, B 0.000, C 0.000 }
gfCNCPoint6[13186] = {X 7.9237, Y 36.6499, Z -8.0000, A 0.000, B 0.000, C 0.000 }
gfCNCPoint6[13187] = {X 8.4177, Y 37.0798, Z -8.0000, A 0.000, B 0.000, C 0.000 }
gfCNCPoint6[13188] = {X 9.2097, Y 37.4820, Z -8.0000, A 0.000, B 0.000, C 0.000 }
gfCNCPoint6[13189] = {X 10.0528, Y 37.7617, Z -8.0000, A 0.000, B 0.000, C 0.000 }
gfCNCPoint6[13190] = {X 11.3578, Y 38.0028, Z -8.0000, A 0.000, B 0.000, C 0.000 }
gfCNCPoint6[13191] = {X 12.6827, Y 38.0782, Z -8.0000, A 0.000, B 0.000, C 0.000 }
gfCNCPoint6[13192] = {X 14.0067, Y 37.9866, Z -8.0000, A 0.000, B 0.000, C 0.000 }
gfCNCPoint6[13193] = {X 15.3086, Y 37.7295, Z -8.0000, A 0.000, B 0.000, C 0.000 }
gfCNCPoint6[13194] = {X 16.5679, Y 37.3109, Z -8.0000, A 0.000, B 0.000, C 0.000 }
gfCNCPoint6[13195] = {X 17.9186, Y 36.6769, Z -8.0000, A 0.000, B 0.000, C 0.000 }
gfCNCPoint6[13196] = {X 19.1915, Y 35.8985, Z -8.0000, A 0.000, B 0.000, C 0.000 }
gfCNCPoint6[13197] = {X 19.2642, Y 35.2210, Z -8.0000, A 0.000, B 0.000, C 0.000 }
gfCNCPoint6[13198] = {X 19.4445, Y 34.5639, Z -8.0000, A 0.000, B 0.000, C 0.000 }
gfCNCPoint6[13199] = {X 19.7278, Y 33.9442, Z -8.0000, A 0.000, B 0.000, C 0.000 }
gfCNCPoint6[13200] = {X 17.9225, Y 34.2667, Z -8.0000, A 0.000, B 0.000, C 0.000 }
gfCNCPoint6[13201] = {X 16.0990, Y 34.4613, Z -8.0000, A 0.000, B 0.000, C 0.000 }
gfCNCPoint6[13202] = {X 15.3745, Y 34.5140, Z -8.0000, A 0.000, B 0.000, C 0.000 }
gfCNCPoint6[13203] = {X 14.6498, Y 34.5646, Z -8.0000, A 0.000, B 0.000, C 0.000 }
gfCNCPoint6[13204] = {X 10.6981, Y 35.1843, Z -8.0000, A 0.000, B 0.000, C 0.000 }
gfCNCPoint6[13205] = {X 18.6436, Y 34.5608, Z -8.0000, A 0.000, B 0.000, C 0.000 }
gfCNCPoint6[13206] = {X 14.6444, Y 34.4848, Z -8.0000, A 0.000, B 0.000, C 0.000 }
gfCNCPoint6[13207] = {X 12.2504, Y 34.6371, Z -8.0000, A 0.000, B 0.000, C 0.000 }
gfCNCPoint6[13208] = {X 9.8551, Y 34.7666, Z -8.0000, A 0.000, B 0.000, C 0.000 }
gfCNCPoint6[13209] = {X 8.6556, Y 34.8680, Z -8.0000, A 0.000, B 0.000, C 0.000 }
gfCNCPoint6[13210] = {X 7.4767, Y 35.1118, Z -8.0000, A 0.000, B 0.000, C 0.000 }
gfCNCPoint6[13211] = {X 7.4298, Y 35.2693, Z -8.0000, A 0.000, B 0.000, C 0.000 }
gfCNCPoint6[13212] = {X 7.4136, Y 35.4329, Z -8.0000, A 0.000, B 0.000, C 0.000 }
gfCNCPoint6[13213] = {X 7.5277, Y 36.1055, Z -8.0000, A 0.000, B 0.000, C 0.000 }
gfCNCPoint6[13214] = {X 7.8616, Y 36.7004, Z -8.0000, A 0.000, B 0.000, C 0.000 }
gfCNCPoint6[13215] = {X 8.3762, Y 37.1483, Z -8.0000, A 0.000, B 0.000, C 0.000 }
gfCNCPoint6[13216] = {X 9.1789, Y 37.5558, Z -8.0000, A 0.000, B 0.000, C 0.000 }
gfCNCPoint6[13217] = {X 10.0333, Y 37.8393, Z -8.0000, A 0.000, B 0.000, C 0.000 }
gfCNCPoint6[13218] = {X 11.3482, Y 38.0823, Z -8.0000, A 0.000, B 0.000, C 0.000 }
gfCNCPoint6[13219] = {X 12.6832, Y 38.1582, Z -8.0000, A 0.000, B 0.000, C 0.000 }
gfCNCPoint6[13220] = {X 14.0172, Y 38.0659, Z -8.0000, A 0.000, B 0.000, C 0.000 }
gfCNCPoint6[13221] = {X 15.3290, Y 37.8068, Z -8.0000, A 0.000, B 0.000, C 0.000 }
gfCNCPoint6[13222] = {X 16.5979, Y 37.3851, Z -8.0000, A 0.000, B 0.000, C 0.000 }
gfCNCPoint6[13223] = {X 17.9745, Y 36.7377, Z -8.0000, A 0.000, B 0.000, C 0.000 }
gfCNCPoint6[13224] = {X 19.2706, Y 35.9411, Z -8.0000, A 0.000, B 0.000, C 0.000 }
gfCNCPoint6[13225] = {X 19.3492, Y 35.2031, Z -8.0000, A 0.000, B 0.000, C 0.000 }
gfCNCPoint6[13226] = {X 19.5577, Y 34.4908, Z -8.0000, A 0.000, B 0.000, C 0.000 }
gfCNCPoint6[13227] = {X 19.8894, Y 33.8270, Z -8.0000, A 0.000, B 0.000, C 0.000 }
gfCNCPoint6[13228] = {X 18.0016, Y 34.1745, Z -8.0000, A 0.000, B 0.000, C 0.000 }
gfCNCPoint6[13229] = {X 16.0932, Y 34.3815, Z -8.0000, A 0.000, B 0.000, C 0.000 }
gfCNCPoint6[13230] = {X 15.3688, Y 34.4342, Z -8.0000, A 0.000, B 0.000, C 0.000 }
gfCNCPoint6[13231] = {X 14.6444, Y 34.4848, Z -8.0000, A 0.000, B 0.000, C 0.000 }
gfCNCPoint6[13232] = {X 10.6927, Y 35.1045, Z -8.0000, A 0.000, B 0.000, C 0.000 }
gfCNCPoint6[13233] = {X 18.6382, Y 34.4809, Z -8.0000, A 0.000, B 0.000, C 0.000 }
gfCNCPoint6[13234] = {X 14.6389, Y 34.4050, Z -8.0000, A 0.000, B 0.000, C 0.000 }
gfCNCPoint6[13235] = {X 12.2462, Y 34.5572, Z -8.0000, A 0.000, B 0.000, C 0.000 }
gfCNCPoint6[13236] = {X 9.8522, Y 34.6866, Z -8.0000, A 0.000, B 0.000, C 0.000 }
gfCNCPoint6[13237] = {X 8.6245, Y 34.7917, Z -8.0000, A 0.000, B 0.000, C 0.000 }
gfCNCPoint6[13238] = {X 7.4185, Y 35.0448, Z -8.0000, A 0.000, B 0.000, C 0.000 }
gfCNCPoint6[13239] = {X 7.3554, Y 35.2342, Z -8.0000, A 0.000, B 0.000, C 0.000 }
gfCNCPoint6[13240] = {X 7.3336, Y 35.4326, Z -8.0000, A 0.000, B 0.000, C 0.000 }
gfCNCPoint6[13241] = {X 7.4002, Y 35.9617, Z -8.0000, A 0.000, B 0.000, C 0.000 }
gfCNCPoint6[13242] = {X 7.5993, Y 36.4565, Z -8.0000, A 0.000, B 0.000, C 0.000 }
gfCNCPoint6[13243] = {X 7.9179, Y 36.8842, Z -8.0000, A 0.000, B 0.000, C 0.000 }
gfCNCPoint6[13244] = {X 8.3348, Y 37.2167, Z -8.0000, A 0.000, B 0.000, C 0.000 }
gfCNCPoint6[13245] = {X 9.1481, Y 37.6296, Z -8.0000, A 0.000, B 0.000, C 0.000 }
gfCNCPoint6[13246] = {X 10.0139, Y 37.9169, Z -8.0000, A 0.000, B 0.000, C 0.000 }
gfCNCPoint6[13247] = {X 11.3387, Y 38.1617, Z -8.0000, A 0.000, B 0.000, C 0.000 }
gfCNCPoint6[13248] = {X 12.6837, Y 38.2382, Z -8.0000, A 0.000, B 0.000, C 0.000 }
gfCNCPoint6[13249] = {X 14.0277, Y 38.1452, Z -8.0000, A 0.000, B 0.000, C 0.000 }
gfCNCPoint6[13250] = {X 15.3494, Y 37.8842, Z -8.0000, A 0.000, B 0.000, C 0.000 }
gfCNCPoint6[13251] = {X 16.6278, Y 37.4593, Z -8.0000, A 0.000, B 0.000, C 0.000 }
gfCNCPoint6[13252] = {X 18.0307, Y 36.7982, Z -8.0000, A 0.000, B 0.000, C 0.000 }
gfCNCPoint6[13253] = {X 19.3501, Y 35.9832, Z -8.0000, A 0.000, B 0.000, C 0.000 }
gfCNCPoint6[13254] = {X 19.4352, Y 35.1815, Z -8.0000, A 0.000, B 0.000, C 0.000 }
gfCNCPoint6[13255] = {X 19.6763, Y 34.4123, Z -8.0000, A 0.000, B 0.000, C 0.000 }
gfCNCPoint6[13256] = {X 20.0639, Y 33.7054, Z -8.0000, A 0.000, B 0.000, C 0.000 }
gfCNCPoint6[13257] = {X 18.0872, Y 34.0809, Z -8.0000, A 0.000, B 0.000, C 0.000 }
gfCNCPoint6[13258] = {X 16.0874, Y 34.3017, Z -8.0000, A 0.000, B 0.000, C 0.000 }
gfCNCPoint6[13259] = {X 15.3632, Y 34.3544, Z -8.0000, A 0.000, B 0.000, C 0.000 }
gfCNCPoint6[13260] = {X 14.6389, Y 34.4050, Z -8.0000, A 0.000, B 0.000, C 0.000 }
gfCNCPoint6[13261] = {X 10.6872, Y 35.0247, Z -8.0000, A 0.000, B 0.000, C 0.000 }
gfCNCPoint6[13262] = {X 14.7699, Y 36.3205, Z -8.0000, A 0.000, B 0.000, C 0.000 }
